    movel(p[new_pose[0], new_pose[1], new_pose[2], current_pose[3], current_pose[4], current_pose[5]], a=1.2, v=0.2000)
    report_progress()
    new_pose = pose_trans(tuft_coords, p[0.8015, 0.1579, -0.0020, 0, 0, 0])
    movel(p[new_pose[0], new_pose[1], new_pose[2], current_pose[3], current_pose[4], current_pose[5]], a=0.8, v=0.2000)
    report_progress()
    set_digital_out(0, True)
    new_pose = pose_trans(tuft_coords, p[0.8015, 0.8921, -0.0020, 0, 0, 0])
    movel(p[new_pose[0], new_pose[1], new_pose[2], current_pose[3], current_pose[4], current_pose[5]], a=1.2, v=0.0600)
    report_progress()
    set_digital_out(0, False)
    new_pose = pose_trans(tuft_coords, p[0.8015, 0.8921, 0.1500, 0, 0, 0])
    movel(p[new_pose[0], new_pose[1], new_pose[2], current_pose[3], current_pose[4], current_pose[5]], a=0.8, v=0.2000)
    report_progress()
    new_pose = pose_trans(tuft_coords, p[0.8035, 0.1579, 0.1500, 0, 0, 0])
    movel(p[new_pose[0], new_pose[1], new_pose[2], current_pose[3], current_pose[4], current_pose[5]], a=1.2, v=0.2000)
    report_progress()
    new_pose = pose_trans(tuft_coords, p[0.8035, 0.1579, -0.0020, 0, 0, 0])
    movel(p[new_pose[0], new_pose[1], new_pose[2], current_pose[3], current_pose[4], current_pose[5]], a=0.8, v=0.2000)
    report_progress()
    set_digital_out(0, True)
    new_pose = pose_trans(tuft_coords, p[0.8035, 0.8921, -0.0020, 0, 0, 0])
    movel(p[new_pose[0], new_pose[1], new_pose[2], current_pose[3], current_pose[4], current_pose[5]], a=1.2, v=0.0600)
    report_progress()
    set_digital_out(0, False)
    new_pose = pose_trans(tuft_coords, p[0.8035, 0.8921, 0.1500, 0, 0, 0])
    movel(p[new_pose[0], new_pose[1], new_pose[2], current_pose[3], current_pose[4], current_pose[5]], a=0.8, v=0.2000)
    report_progress()
    new_pose = pose_trans(tuft_coords, p[0.8054, 0.1579, 0.1500, 0, 0, 0])
    movel(p[new_pose[0], new_pose[1], new_pose[2], current_pose[3], current_pose[4], current_pose[5]], a=1.2, v=0.2000)
    report_progress()
    new_pose = pose_trans(tuft_coords, p[0.8054, 0.1579, -0.0020, 0, 0, 0])
    movel(p[new_pose[0], new_pose[1], new_pose[2], current_pose[3], current_pose[4], current_pose[5]], a=0.8, v=0.2000)
    report_progress()
    set_digital_out(0, True)
    new_pose = pose_trans(tuft_coords, p[0.8054, 0.8921, -0.0020, 0, 0, 0])
    movel(p[new_pose[0], new_pose[1], new_pose[2], current_pose[3], current_pose[4], current_pose[5]], a=1.2, v=0.0600)
    report_progress()
    set_digital_out(0, False)
    new_pose = pose_trans(tuft_coords, p[0.8054, 0.8921, 0.1500, 0, 0, 0])
    movel(p[new_pose[0], new_pose[1], new_pose[2], current_pose[3], current_pose[4], current_pose[5]], a=0.8, v=0.2000)
    report_progress()
    new_pose = pose_trans(tuft_coords, p[0.8074, 0.1598, 0.1500, 0, 0, 0])
    movel(p[new_pose[0], new_pose[1], new_pose[2], current_pose[3], current_pose[4], current_pose[5]], a=1.2, v=0.2000)
    report_progress()
    new_pose = pose_trans(tuft_coords, p[0.8074, 0.1598, -0.0020, 0, 0, 0])
    movel(p[new_pose[0], new_pose[1], new_pose[2], current_pose[3], current_pose[4], current_pose[5]], a=0.8, v=0.2000)
    report_progress()
    set_digital_out(0, True)
    new_pose = pose_trans(tuft_coords, p[0.8074, 0.8902, -0.0020, 0, 0, 0])
    movel(p[new_pose[0], new_pose[1], new_pose[2], current_pose[3], current_pose[4], current_pose[5]], a=1.2, v=0.0600)
    report_progress()
    set_digital_out(0, False)
    new_pose = pose_trans(tuft_coords, p[0.8074, 0.8902, 0.1500, 0, 0, 0])
    movel(p[new_pose[0], new_pose[1], new_pose[2], current_pose[3], current_pose[4], current_pose[5]], a=0.8, v=0.2000)
    report_progress()
    new_pose = pose_trans(tuft_coords, p[0.8093, 0.1598, 0.1500, 0, 0, 0])
    movel(p[new_pose[0], new_pose[1], new_pose[2], current_pose[3], current_pose[4], current_pose[5]], a=1.2, v=0.2000)
    report_progress()
    new_pose = pose_trans(tuft_coords, p[0.8093, 0.1598, -0.0020, 0, 0, 0])
    movel(p[new_pose[0], new_pose[1], new_pose[2], current_pose[3], current_pose[4], current_pose[5]], a=0.8, v=0.2000)
    report_progress()
    set_digital_out(0, True)
    new_pose = pose_trans(tuft_coords, p[0.8093, 0.8902, -0.0020, 0, 0, 0])
    movel(p[new_pose[0], new_pose[1], new_pose[2], current_pose[3], current_pose[4], current_pose[5]], a=1.2, v=0.0600)
    report_progress()
    set_digital_out(0, False)
    new_pose = pose_trans(tuft_coords, p[0.8093, 0.8902, 0.1500, 0, 0, 0])
    movel(p[new_pose[0], new_pose[1], new_pose[2], current_pose[3], current_pose[4], current_pose[5]], a=0.8, v=0.2000)
    report_progress()
    new_pose = pose_trans(tuft_coords, p[0.8113, 0.1598, 0.1500, 0, 0, 0])
    movel(p[new_pose[0], new_pose[1], new_pose[2], current_pose[3], current_pose[4], current_pose[5]], a=1.2, v=0.2000)
    report_progress()
    new_pose = pose_trans(tuft_coords, p[0.8113, 0.1598, -0.0020, 0, 0, 0])
    movel(p[new_pose[0], new_pose[1], new_pose[2], current_pose[3], current_pose[4], current_pose[5]], a=0.8, v=0.2000)
    report_progress()
    set_digital_out(0, True)
    new_pose = pose_trans(tuft_coords, p[0.8113, 0.8902, -0.0020, 0, 0, 0])
    movel(p[new_pose[0], new_pose[1], new_pose[2], current_pose[3], current_pose[4], current_pose[5]], a=1.2, v=0.0600)
    report_progress()
    set_digital_out(0, False)
    new_pose = pose_trans(tuft_coords, p[0.8113, 0.8902, 0.1500, 0, 0, 0])
    movel(p[new_pose[0], new_pose[1], new_pose[2], current_pose[3], current_pose[4], current_pose[5]], a=0.8, v=0.2000)
    report_progress()
    new_pose = pose_trans(tuft_coords, p[0.8132, 0.1598, 0.1500, 0, 0, 0])
    movel(p[new_pose[0], new_pose[1], new_pose[2], current_pose[3], current_pose[4], current_pose[5]], a=1.2, v=0.2000)
    report_progress()
    new_pose = pose_trans(tuft_coords, p[0.8132, 0.1598, -0.0020, 0, 0, 0])
    movel(p[new_pose[0], new_pose[1], new_pose[2], current_pose[3], current_pose[4], current_pose[5]], a=0.8, v=0.2000)
    report_progress()
    set_digital_out(0, True)
    new_pose = pose_trans(tuft_coords, p[0.8132, 0.8902, -0.0020, 0, 0, 0])
    movel(p[new_pose[0], new_pose[1], new_pose[2], current_pose[3], current_pose[4], current_pose[5]], a=1.2, v=0.0600)
    report_progress()
    set_digital_out(0, False)
    new_pose = pose_trans(tuft_coords, p[0.8132, 0.8902, 0.1500, 0, 0, 0])
    movel(p[new_pose[0], new_pose[1], new_pose[2], current_pose[3], current_pose[4], current_pose[5]], a=0.8, v=0.2000)
    report_progress()
    new_pose = pose_trans(tuft_coords, p[0.8151, 0.1598, 0.1500, 0, 0, 0])
    movel(p[new_pose[0], new_pose[1], new_pose[2], current_pose[3], current_pose[4], current_pose[5]], a=1.2, v=0.2000)
    report_progress()
    new_pose = pose_trans(tuft_coords, p[0.8151, 0.1598, -0.0020, 0, 0, 0])
    movel(p[new_pose[0], new_pose[1], new_pose[2], current_pose[3], current_pose[4], current_pose[5]], a=0.8, v=0.2000)
    report_progress()
    set_digital_out(0, True)
    new_pose = pose_trans(tuft_coords, p[0.8151, 0.8902, -0.0020, 0, 0, 0])
    movel(p[new_pose[0], new_pose[1], new_pose[2], current_pose[3], current_pose[4], current_pose[5]], a=1.2, v=0.0600)
    report_progress()
    set_digital_out(0, False)
    new_pose = pose_trans(tuft_coords, p[0.8151, 0.8902, 0.1500, 0, 0, 0])
    movel(p[new_pose[0], new_pose[1], new_pose[2], current_pose[3], current_pose[4], current_pose[5]], a=0.8, v=0.2000)
    report_progress()
    new_pose = pose_trans(tuft_coords, p[0.8171, 0.1598, 0.1500, 0, 0, 0])
    movel(p[new_pose[0], new_pose[1], new_pose[2], current_pose[3], current_pose[4], current_pose[5]], a=1.2, v=0.2000)
    report_progress()
    new_pose = pose_trans(tuft_coords, p[0.8171, 0.1598, -0.0020, 0, 0, 0])
    movel(p[new_pose[0], new_pose[1], new_pose[2], current_pose[3], current_pose[4], current_pose[5]], a=0.8, v=0.2000)
    report_progress()
    set_digital_out(0, True)
    new_pose = pose_trans(tuft_coords, p[0.8171, 0.8902, -0.0020, 0, 0, 0])
    movel(p[new_pose[0], new_pose[1], new_pose[2], current_pose[3], current_pose[4], current_pose[5]], a=1.2, v=0.0600)
    report_progress()
    set_digital_out(0, False)
    new_pose = pose_trans(tuft_coords, p[0.8171, 0.8902, 0.1500, 0, 0, 0])
    movel(p[new_pose[0], new_pose[1], new_pose[2], current_pose[3], current_pose[4], current_pose[5]], a=0.8, v=0.2000)
    report_progress()
    new_pose = pose_trans(tuft_coords, p[0.8190, 0.1618, 0.1500, 0, 0, 0])
    movel(p[new_pose[0], new_pose[1], new_pose[2], current_pose[3], current_pose[4], current_pose[5]], a=1.2, v=0.2000)
    report_progress()
    new_pose = pose_trans(tuft_coords, p[0.8190, 0.1618, -0.0020, 0, 0, 0])
    movel(p[new_pose[0], new_pose[1], new_pose[2], current_pose[3], current_pose[4], current_pose[5]], a=0.8, v=0.2000)
    report_progress()
    set_digital_out(0, True)
    new_pose = pose_trans(tuft_coords, p[0.8190, 0.8882, -0.0020, 0, 0, 0])
    movel(p[new_pose[0], new_pose[1], new_pose[2], current_pose[3], current_pose[4], current_pose[5]], a=1.2, v=0.0600)
    report_progress()
    set_digital_out(0, False)
    new_pose = pose_trans(tuft_coords, p[0.8190, 0.8882, 0.1500, 0, 0, 0])
    movel(p[new_pose[0], new_pose[1], new_pose[2], current_pose[3], current_pose[4], current_pose[5]], a=0.8, v=0.2000)
    report_progress()
    new_pose = pose_trans(tuft_coords, p[0.8210, 0.1618, 0.1500, 0, 0, 0])
    movel(p[new_pose[0], new_pose[1], new_pose[2], current_pose[3], current_pose[4], current_pose[5]], a=1.2, v=0.2000)
    report_progress()
    new_pose = pose_trans(tuft_coords, p[0.8210, 0.1618, -0.0020, 0, 0, 0])
    movel(p[new_pose[0], new_pose[1], new_pose[2], current_pose[3], current_pose[4], current_pose[5]], a=0.8, v=0.2000)
    report_progress()
    set_digital_out(0, True)
    new_pose = pose_trans(tuft_coords, p[0.8210, 0.8882, -0.0020, 0, 0, 0])
    movel(p[new_pose[0], new_pose[1], new_pose[2], current_pose[3], current_pose[4], current_pose[5]], a=1.2, v=0.0600)
    report_progress()
    set_digital_out(0, False)
    new_pose = pose_trans(tuft_coords, p[0.8210, 0.8882, 0.1500, 0, 0, 0])
    movel(p[new_pose[0], new_pose[1], new_pose[2], current_pose[3], current_pose[4], current_pose[5]], a=0.8, v=0.2000)
    report_progress()
    new_pose = pose_trans(tuft_coords, p[0.8229, 0.1618, 0.1500, 0, 0, 0])
    movel(p[new_pose[0], new_pose[1], new_pose[2], current_pose[3], current_pose[4], current_pose[5]], a=1.2, v=0.2000)
    report_progress()
    new_pose = pose_trans(tuft_coords, p[0.8229, 0.1618, -0.0020, 0, 0, 0])
    movel(p[new_pose[0], new_pose[1], new_pose[2], current_pose[3], current_pose[4], current_pose[5]], a=0.8, v=0.2000)
    report_progress()
    set_digital_out(0, True)
    new_pose = pose_trans(tuft_coords, p[0.8229, 0.8882, -0.0020, 0, 0, 0])
    movel(p[new_pose[0], new_pose[1], new_pose[2], current_pose[3], current_pose[4], current_pose[5]], a=1.2, v=0.0600)
    report_progress()
    set_digital_out(0, False)
    new_pose = pose_trans(tuft_coords, p[0.8229, 0.8882, 0.1500, 0, 0, 0])
    movel(p[new_pose[0], new_pose[1], new_pose[2], current_pose[3], current_pose[4], current_pose[5]], a=0.8, v=0.2000)
    report_progress()
    new_pose = pose_trans(tuft_coords, p[0.8249, 0.1618, 0.1500, 0, 0, 0])
    movel(p[new_pose[0], new_pose[1], new_pose[2], current_pose[3], current_pose[4], current_pose[5]], a=1.2, v=0.2000)
    report_progress()
    new_pose = pose_trans(tuft_coords, p[0.8249, 0.1618, -0.0020, 0, 0, 0])
    movel(p[new_pose[0], new_pose[1], new_pose[2], current_pose[3], current_pose[4], current_pose[5]], a=0.8, v=0.2000)
    report_progress()
    set_digital_out(0, True)
    new_pose = pose_trans(tuft_coords, p[0.8249, 0.8882, -0.0020, 0, 0, 0])
    movel(p[new_pose[0], new_pose[1], new_pose[2], current_pose[3], current_pose[4], current_pose[5]], a=1.2, v=0.0600)
    report_progress()
    set_digital_out(0, False)
    new_pose = pose_trans(tuft_coords, p[0.8249, 0.8882, 0.1500, 0, 0, 0])
    movel(p[new_pose[0], new_pose[1], new_pose[2], current_pose[3], current_pose[4], current_pose[5]], a=0.8, v=0.2000)
    report_progress()
    new_pose = pose_trans(tuft_coords, p[0.8268, 0.1618, 0.1500, 0, 0, 0])
    movel(p[new_pose[0], new_pose[1], new_pose[2], current_pose[3], current_pose[4], current_pose[5]], a=1.2, v=0.2000)
    report_progress()
    new_pose = pose_trans(tuft_coords, p[0.8268, 0.1618, -0.0020, 0, 0, 0])
    movel(p[new_pose[0], new_pose[1], new_pose[2], current_pose[3], current_pose[4], current_pose[5]], a=0.8, v=0.2000)
    report_progress()
    set_digital_out(0, True)
    new_pose = pose_trans(tuft_coords, p[0.8268, 0.8882, -0.0020, 0, 0, 0])
    movel(p[new_pose[0], new_pose[1], new_pose[2], current_pose[3], current_pose[4], current_pose[5]], a=1.2, v=0.0600)
    report_progress()
    set_digital_out(0, False)
    new_pose = pose_trans(tuft_coords, p[0.8268, 0.8882, 0.1500, 0, 0, 0])
    movel(p[new_pose[0], new_pose[1], new_pose[2], current_pose[3], current_pose[4], current_pose[5]], a=0.8, v=0.2000)
    report_progress()
    new_pose = pose_trans(tuft_coords, p[0.8287, 0.1638, 0.1500, 0, 0, 0])
    movel(p[new_pose[0], new_pose[1], new_pose[2], current_pose[3], current_pose[4], current_pose[5]], a=1.2, v=0.2000)
    report_progress()
    new_pose = pose_trans(tuft_coords, p[0.8287, 0.1638, -0.0020, 0, 0, 0])
    movel(p[new_pose[0], new_pose[1], new_pose[2], current_pose[3], current_pose[4], current_pose[5]], a=0.8, v=0.2000)
    report_progress()
    set_digital_out(0, True)
    new_pose = pose_trans(tuft_coords, p[0.8287, 0.8862, -0.0020, 0, 0, 0])
    movel(p[new_pose[0], new_pose[1], new_pose[2], current_pose[3], current_pose[4], current_pose[5]], a=1.2, v=0.0600)
    report_progress()
    set_digital_out(0, False)
    new_pose = pose_trans(tuft_coords, p[0.8287, 0.8862, 0.1500, 0, 0, 0])
    movel(p[new_pose[0], new_pose[1], new_pose[2], current_pose[3], current_pose[4], current_pose[5]], a=0.8, v=0.2000)
    report_progress()
    new_pose = pose_trans(tuft_coords, p[0.8307, 0.1638, 0.1500, 0, 0, 0])
    movel(p[new_pose[0], new_pose[1], new_pose[2], current_pose[3], current_pose[4], current_pose[5]], a=1.2, v=0.2000)
    report_progress()
    new_pose = pose_trans(tuft_coords, p[0.8307, 0.1638, -0.0020, 0, 0, 0])
    movel(p[new_pose[0], new_pose[1], new_pose[2], current_pose[3], current_pose[4], current_pose[5]], a=0.8, v=0.2000)
    report_progress()
    set_digital_out(0, True)
    new_pose = pose_trans(tuft_coords, p[0.8307, 0.8862, -0.0020, 0, 0, 0])
    movel(p[new_pose[0], new_pose[1], new_pose[2], current_pose[3], current_pose[4], current_pose[5]], a=1.2, v=0.0600)
    report_progress()
    set_digital_out(0, False)
    new_pose = pose_trans(tuft_coords, p[0.8307, 0.8862, 0.1500, 0, 0, 0])
    movel(p[new_pose[0], new_pose[1], new_pose[2], current_pose[3], current_pose[4], current_pose[5]], a=0.8, v=0.2000)
    report_progress()
    new_pose = pose_trans(tuft_coords, p[0.8326, 0.1638, 0.1500, 0, 0, 0])
    movel(p[new_pose[0], new_pose[1], new_pose[2], current_pose[3], current_pose[4], current_pose[5]], a=1.2, v=0.2000)
    report_progress()
    new_pose = pose_trans(tuft_coords, p[0.8326, 0.1638, -0.0020, 0, 0, 0])
    movel(p[new_pose[0], new_pose[1], new_pose[2], current_pose[3], current_pose[4], current_pose[5]], a=0.8, v=0.2000)
    report_progress()
    set_digital_out(0, True)
    new_pose = pose_trans(tuft_coords, p[0.8326, 0.8862, -0.0020, 0, 0, 0])
    movel(p[new_pose[0], new_pose[1], new_pose[2], current_pose[3], current_pose[4], current_pose[5]], a=1.2, v=0.0600)
    report_progress()
    set_digital_out(0, False)
    new_pose = pose_trans(tuft_coords, p[0.8326, 0.8862, 0.1500, 0, 0, 0])
    movel(p[new_pose[0], new_pose[1], new_pose[2], current_pose[3], current_pose[4], current_pose[5]], a=0.8, v=0.2000)
    report_progress()
    new_pose = pose_trans(tuft_coords, p[0.8346, 0.1638, 0.1500, 0, 0, 0])
    movel(p[new_pose[0], new_pose[1], new_pose[2], current_pose[3], current_pose[4], current_pose[5]], a=1.2, v=0.2000)
    report_progress()
    new_pose = pose_trans(tuft_coords, p[0.8346, 0.1638, -0.0020, 0, 0, 0])
    movel(p[new_pose[0], new_pose[1], new_pose[2], current_pose[3], current_pose[4], current_pose[5]], a=0.8, v=0.2000)
    report_progress()
    set_digital_out(0, True)
    new_pose = pose_trans(tuft_coords, p[0.8346, 0.8862, -0.0020, 0, 0, 0])
    movel(p[new_pose[0], new_pose[1], new_pose[2], current_pose[3], current_pose[4], current_pose[5]], a=1.2, v=0.0600)
    report_progress()
    set_digital_out(0, False)
    new_pose = pose_trans(tuft_coords, p[0.8346, 0.8862, 0.1500, 0, 0, 0])
    movel(p[new_pose[0], new_pose[1], new_pose[2], current_pose[3], current_pose[4], current_pose[5]], a=0.8, v=0.2000)
    report_progress()
    new_pose = pose_trans(tuft_coords, p[0.8365, 0.1658, 0.1500, 0, 0, 0])
    movel(p[new_pose[0], new_pose[1], new_pose[2], current_pose[3], current_pose[4], current_pose[5]], a=1.2, v=0.2000)
    report_progress()
    new_pose = pose_trans(tuft_coords, p[0.8365, 0.1658, -0.0020, 0, 0, 0])
    movel(p[new_pose[0], new_pose[1], new_pose[2], current_pose[3], current_pose[4], current_pose[5]], a=0.8, v=0.2000)
    report_progress()
    set_digital_out(0, True)
    new_pose = pose_trans(tuft_coords, p[0.8365, 0.8842, -0.0020, 0, 0, 0])
    movel(p[new_pose[0], new_pose[1], new_pose[2], current_pose[3], current_pose[4], current_pose[5]], a=1.2, v=0.0600)
    report_progress()
    set_digital_out(0, False)
    new_pose = pose_trans(tuft_coords, p[0.8365, 0.8842, 0.1500, 0, 0, 0])
    movel(p[new_pose[0], new_pose[1], new_pose[2], current_pose[3], current_pose[4], current_pose[5]], a=0.8, v=0.2000)
    report_progress()
    new_pose = pose_trans(tuft_coords, p[0.8385, 0.1658, 0.1500, 0, 0, 0])
    movel(p[new_pose[0], new_pose[1], new_pose[2], current_pose[3], current_pose[4], current_pose[5]], a=1.2, v=0.2000)
    report_progress()
    new_pose = pose_trans(tuft_coords, p[0.8385, 0.1658, -0.0020, 0, 0, 0])
    movel(p[new_pose[0], new_pose[1], new_pose[2], current_pose[3], current_pose[4], current_pose[5]], a=0.8, v=0.2000)
    report_progress()
    set_digital_out(0, True)
    new_pose = pose_trans(tuft_coords, p[0.8385, 0.8842, -0.0020, 0, 0, 0])
    movel(p[new_pose[0], new_pose[1], new_pose[2], current_pose[3], current_pose[4], current_pose[5]], a=1.2, v=0.0600)
    report_progress()
    set_digital_out(0, False)
    new_pose = pose_trans(tuft_coords, p[0.8385, 0.8842, 0.1500, 0, 0, 0])
    movel(p[new_pose[0], new_pose[1], new_pose[2], current_pose[3], current_pose[4], current_pose[5]], a=0.8, v=0.2000)
    report_progress()
    new_pose = pose_trans(tuft_coords, p[0.8404, 0.1658, 0.1500, 0, 0, 0])
    movel(p[new_pose[0], new_pose[1], new_pose[2], current_pose[3], current_pose[4], current_pose[5]], a=1.2, v=0.2000)
    report_progress()
    new_pose = pose_trans(tuft_coords, p[0.8404, 0.1658, -0.0020, 0, 0, 0])
    movel(p[new_pose[0], new_pose[1], new_pose[2], current_pose[3], current_pose[4], current_pose[5]], a=0.8, v=0.2000)
    report_progress()
    set_digital_out(0, True)
    new_pose = pose_trans(tuft_coords, p[0.8404, 0.8842, -0.0020, 0, 0, 0])
    movel(p[new_pose[0], new_pose[1], new_pose[2], current_pose[3], current_pose[4], current_pose[5]], a=1.2, v=0.0600)
    report_progress()
    set_digital_out(0, False)
    new_pose = pose_trans(tuft_coords, p[0.8404, 0.8842, 0.1500, 0, 0, 0])
    movel(p[new_pose[0], new_pose[1], new_pose[2], current_pose[3], current_pose[4], current_pose[5]], a=0.8, v=0.2000)
    report_progress()
    new_pose = pose_trans(tuft_coords, p[0.8424, 0.1658, 0.1500, 0, 0, 0])
    movel(p[new_pose[0], new_pose[1], new_pose[2], current_pose[3], current_pose[4], current_pose[5]], a=1.2, v=0.2000)
    report_progress()
    new_pose = pose_trans(tuft_coords, p[0.8424, 0.1658, -0.0020, 0, 0, 0])
    movel(p[new_pose[0], new_pose[1], new_pose[2], current_pose[3], current_pose[4], current_pose[5]], a=0.8, v=0.2000)
    report_progress()
    set_digital_out(0, True)
    new_pose = pose_trans(tuft_coords, p[0.8424, 0.8842, -0.0020, 0, 0, 0])
    movel(p[new_pose[0], new_pose[1], new_pose[2], current_pose[3], current_pose[4], current_pose[5]], a=1.2, v=0.0600)
    report_progress()
    set_digital_out(0, False)
    new_pose = pose_trans(tuft_coords, p[0.8424, 0.8842, 0.1500, 0, 0, 0])
    movel(p[new_pose[0], new_pose[1], new_pose[2], current_pose[3], current_pose[4], current_pose[5]], a=0.8, v=0.2000)
    report_progress()
    new_pose = pose_trans(tuft_coords, p[0.8443, 0.1678, 0.1500, 0, 0, 0])
    movel(p[new_pose[0], new_pose[1], new_pose[2], current_pose[3], current_pose[4], current_pose[5]], a=1.2, v=0.2000)
    report_progress()
    new_pose = pose_trans(tuft_coords, p[0.8443, 0.1678, -0.0020, 0, 0, 0])
    movel(p[new_pose[0], new_pose[1], new_pose[2], current_pose[3], current_pose[4], current_pose[5]], a=0.8, v=0.2000)
    report_progress()
    set_digital_out(0, True)
    new_pose = pose_trans(tuft_coords, p[0.8443, 0.8822, -0.0020, 0, 0, 0])
    movel(p[new_pose[0], new_pose[1], new_pose[2], current_pose[3], current_pose[4], current_pose[5]], a=1.2, v=0.0600)
    report_progress()
    set_digital_out(0, False)
    new_pose = pose_trans(tuft_coords, p[0.8443, 0.8822, 0.1500, 0, 0, 0])
    movel(p[new_pose[0], new_pose[1], new_pose[2], current_pose[3], current_pose[4], current_pose[5]], a=0.8, v=0.2000)
    report_progress()
    new_pose = pose_trans(tuft_coords, p[0.8462, 0.1678, 0.1500, 0, 0, 0])
    movel(p[new_pose[0], new_pose[1], new_pose[2], current_pose[3], current_pose[4], current_pose[5]], a=1.2, v=0.2000)
    report_progress()
    new_pose = pose_trans(tuft_coords, p[0.8462, 0.1678, -0.0020, 0, 0, 0])
    movel(p[new_pose[0], new_pose[1], new_pose[2], current_pose[3], current_pose[4], current_pose[5]], a=0.8, v=0.2000)
    report_progress()
    set_digital_out(0, True)
    new_pose = pose_trans(tuft_coords, p[0.8462, 0.8822, -0.0020, 0, 0, 0])
    movel(p[new_pose[0], new_pose[1], new_pose[2], current_pose[3], current_pose[4], current_pose[5]], a=1.2, v=0.0600)
    report_progress()
    set_digital_out(0, False)
    new_pose = pose_trans(tuft_coords, p[0.8462, 0.8822, 0.1500, 0, 0, 0])
    movel(p[new_pose[0], new_pose[1], new_pose[2], current_pose[3], current_pose[4], current_pose[5]], a=0.8, v=0.2000)
    report_progress()
    new_pose = pose_trans(tuft_coords, p[0.8482, 0.1678, 0.1500, 0, 0, 0])
    movel(p[new_pose[0], new_pose[1], new_pose[2], current_pose[3], current_pose[4], current_pose[5]], a=1.2, v=0.2000)
    report_progress()
    new_pose = pose_trans(tuft_coords, p[0.8482, 0.1678, -0.0020, 0, 0, 0])
    movel(p[new_pose[0], new_pose[1], new_pose[2], current_pose[3], current_pose[4], current_pose[5]], a=0.8, v=0.2000)
    report_progress()
    set_digital_out(0, True)
    new_pose = pose_trans(tuft_coords, p[0.8482, 0.8822, -0.0020, 0, 0, 0])
    movel(p[new_pose[0], new_pose[1], new_pose[2], current_pose[3], current_pose[4], current_pose[5]], a=1.2, v=0.0600)
    report_progress()
    set_digital_out(0, False)
    new_pose = pose_trans(tuft_coords, p[0.8482, 0.8822, 0.1500, 0, 0, 0])
    movel(p[new_pose[0], new_pose[1], new_pose[2], current_pose[3], current_pose[4], current_pose[5]], a=0.8, v=0.2000)
    report_progress()
    new_pose = pose_trans(tuft_coords, p[0.8501, 0.1678, 0.1500, 0, 0, 0])
    movel(p[new_pose[0], new_pose[1], new_pose[2], current_pose[3], current_pose[4], current_pose[5]], a=1.2, v=0.2000)
    report_progress()
    new_pose = pose_trans(tuft_coords, p[0.8501, 0.1678, -0.0020, 0, 0, 0])
    movel(p[new_pose[0], new_pose[1], new_pose[2], current_pose[3], current_pose[4], current_pose[5]], a=0.8, v=0.2000)
    report_progress()
    set_digital_out(0, True)
    new_pose = pose_trans(tuft_coords, p[0.8501, 0.8822, -0.0020, 0, 0, 0])
    movel(p[new_pose[0], new_pose[1], new_pose[2], current_pose[3], current_pose[4], current_pose[5]], a=1.2, v=0.0600)
    report_progress()
    set_digital_out(0, False)
    new_pose = pose_trans(tuft_coords, p[0.8501, 0.8822, 0.1500, 0, 0, 0])
    movel(p[new_pose[0], new_pose[1], new_pose[2], current_pose[3], current_pose[4], current_pose[5]], a=0.8, v=0.2000)
    report_progress()
    new_pose = pose_trans(tuft_coords, p[0.8521, 0.1697, 0.1500, 0, 0, 0])
    movel(p[new_pose[0], new_pose[1], new_pose[2], current_pose[3], current_pose[4], current_pose[5]], a=1.2, v=0.2000)
    report_progress()
    new_pose = pose_trans(tuft_coords, p[0.8521, 0.1697, -0.0020, 0, 0, 0])
    movel(p[new_pose[0], new_pose[1], new_pose[2], current_pose[3], current_pose[4], current_pose[5]], a=0.8, v=0.2000)
    report_progress()
    set_digital_out(0, True)
    new_pose = pose_trans(tuft_coords, p[0.8521, 0.8803, -0.0020, 0, 0, 0])
    movel(p[new_pose[0], new_pose[1], new_pose[2], current_pose[3], current_pose[4], current_pose[5]], a=1.2, v=0.0600)
    report_progress()
    set_digital_out(0, False)
    new_pose = pose_trans(tuft_coords, p[0.8521, 0.8803, 0.1500, 0, 0, 0])
    movel(p[new_pose[0], new_pose[1], new_pose[2], current_pose[3], current_pose[4], current_pose[5]], a=0.8, v=0.2000)
    report_progress()
    new_pose = pose_trans(tuft_coords, p[0.8540, 0.1697, 0.1500, 0, 0, 0])
    movel(p[new_pose[0], new_pose[1], new_pose[2], current_pose[3], current_pose[4], current_pose[5]], a=1.2, v=0.2000)
    report_progress()
    new_pose = pose_trans(tuft_coords, p[0.8540, 0.1697, -0.0020, 0, 0, 0])
    movel(p[new_pose[0], new_pose[1], new_pose[2], current_pose[3], current_pose[4], current_pose[5]], a=0.8, v=0.2000)
    report_progress()
    set_digital_out(0, True)
    new_pose = pose_trans(tuft_coords, p[0.8540, 0.8803, -0.0020, 0, 0, 0])
    movel(p[new_pose[0], new_pose[1], new_pose[2], current_pose[3], current_pose[4], current_pose[5]], a=1.2, v=0.0600)
    report_progress()
    set_digital_out(0, False)
    new_pose = pose_trans(tuft_coords, p[0.8540, 0.8803, 0.1500, 0, 0, 0])
    movel(p[new_pose[0], new_pose[1], new_pose[2], current_pose[3], current_pose[4], current_pose[5]], a=0.8, v=0.2000)
    report_progress()
    new_pose = pose_trans(tuft_coords, p[0.8560, 0.1697, 0.1500, 0, 0, 0])
    movel(p[new_pose[0], new_pose[1], new_pose[2], current_pose[3], current_pose[4], current_pose[5]], a=1.2, v=0.2000)
    report_progress()
    new_pose = pose_trans(tuft_coords, p[0.8560, 0.1697, -0.0020, 0, 0, 0])
    movel(p[new_pose[0], new_pose[1], new_pose[2], current_pose[3], current_pose[4], current_pose[5]], a=0.8, v=0.2000)
    report_progress()
    set_digital_out(0, True)
    new_pose = pose_trans(tuft_coords, p[0.8560, 0.8803, -0.0020, 0, 0, 0])
    movel(p[new_pose[0], new_pose[1], new_pose[2], current_pose[3], current_pose[4], current_pose[5]], a=1.2, v=0.0600)
    report_progress()
    set_digital_out(0, False)
    new_pose = pose_trans(tuft_coords, p[0.8560, 0.8803, 0.1500, 0, 0, 0])
    movel(p[new_pose[0], new_pose[1], new_pose[2], current_pose[3], current_pose[4], current_pose[5]], a=0.8, v=0.2000)
    report_progress()
    new_pose = pose_trans(tuft_coords, p[0.8579, 0.1717, 0.1500, 0, 0, 0])
    movel(p[new_pose[0], new_pose[1], new_pose[2], current_pose[3], current_pose[4], current_pose[5]], a=1.2, v=0.2000)
    report_progress()
    new_pose = pose_trans(tuft_coords, p[0.8579, 0.1717, -0.0020, 0, 0, 0])
    movel(p[new_pose[0], new_pose[1], new_pose[2], current_pose[3], current_pose[4], current_pose[5]], a=0.8, v=0.2000)
    report_progress()
    set_digital_out(0, True)
    new_pose = pose_trans(tuft_coords, p[0.8579, 0.8783, -0.0020, 0, 0, 0])
    movel(p[new_pose[0], new_pose[1], new_pose[2], current_pose[3], current_pose[4], current_pose[5]], a=1.2, v=0.0600)
    report_progress()
    set_digital_out(0, False)
    new_pose = pose_trans(tuft_coords, p[0.8579, 0.8783, 0.1500, 0, 0, 0])
    movel(p[new_pose[0], new_pose[1], new_pose[2], current_pose[3], current_pose[4], current_pose[5]], a=0.8, v=0.2000)
    report_progress()
    new_pose = pose_trans(tuft_coords, p[0.8599, 0.1717, 0.1500, 0, 0, 0])
    movel(p[new_pose[0], new_pose[1], new_pose[2], current_pose[3], current_pose[4], current_pose[5]], a=1.2, v=0.2000)
    report_progress()
    new_pose = pose_trans(tuft_coords, p[0.8599, 0.1717, -0.0020, 0, 0, 0])
    movel(p[new_pose[0], new_pose[1], new_pose[2], current_pose[3], current_pose[4], current_pose[5]], a=0.8, v=0.2000)
    report_progress()
    set_digital_out(0, True)
    new_pose = pose_trans(tuft_coords, p[0.8599, 0.8783, -0.0020, 0, 0, 0])
    movel(p[new_pose[0], new_pose[1], new_pose[2], current_pose[3], current_pose[4], current_pose[5]], a=1.2, v=0.0600)
    report_progress()
    set_digital_out(0, False)
    new_pose = pose_trans(tuft_coords, p[0.8599, 0.8783, 0.1500, 0, 0, 0])
    movel(p[new_pose[0], new_pose[1], new_pose[2], current_pose[3], current_pose[4], current_pose[5]], a=0.8, v=0.2000)
    report_progress()
    new_pose = pose_trans(tuft_coords, p[0.8618, 0.1717, 0.1500, 0, 0, 0])
    movel(p[new_pose[0], new_pose[1], new_pose[2], current_pose[3], current_pose[4], current_pose[5]], a=1.2, v=0.2000)
    report_progress()
    new_pose = pose_trans(tuft_coords, p[0.8618, 0.1717, -0.0020, 0, 0, 0])
    movel(p[new_pose[0], new_pose[1], new_pose[2], current_pose[3], current_pose[4], current_pose[5]], a=0.8, v=0.2000)
    report_progress()
    set_digital_out(0, True)
    new_pose = pose_trans(tuft_coords, p[0.8618, 0.8783, -0.0020, 0, 0, 0])
    movel(p[new_pose[0], new_pose[1], new_pose[2], current_pose[3], current_pose[4], current_pose[5]], a=1.2, v=0.0600)
    report_progress()
    set_digital_out(0, False)
    new_pose = pose_trans(tuft_coords, p[0.8618, 0.8783, 0.1500, 0, 0, 0])
    movel(p[new_pose[0], new_pose[1], new_pose[2], current_pose[3], current_pose[4], current_pose[5]], a=0.8, v=0.2000)
    report_progress()
    new_pose = pose_trans(tuft_coords, p[0.8638, 0.1737, 0.1500, 0, 0, 0])
    movel(p[new_pose[0], new_pose[1], new_pose[2], current_pose[3], current_pose[4], current_pose[5]], a=1.2, v=0.2000)
    report_progress()
    new_pose = pose_trans(tuft_coords, p[0.8638, 0.1737, -0.0020, 0, 0, 0])
    movel(p[new_pose[0], new_pose[1], new_pose[2], current_pose[3], current_pose[4], current_pose[5]], a=0.8, v=0.2000)
    report_progress()
    set_digital_out(0, True)
    new_pose = pose_trans(tuft_coords, p[0.8638, 0.8763, -0.0020, 0, 0, 0])
    movel(p[new_pose[0], new_pose[1], new_pose[2], current_pose[3], current_pose[4], current_pose[5]], a=1.2, v=0.0600)
    report_progress()
    set_digital_out(0, False)
    new_pose = pose_trans(tuft_coords, p[0.8638, 0.8763, 0.1500, 0, 0, 0])
    movel(p[new_pose[0], new_pose[1], new_pose[2], current_pose[3], current_pose[4], current_pose[5]], a=0.8, v=0.2000)
    report_progress()
    new_pose = pose_trans(tuft_coords, p[0.8657, 0.1737, 0.1500, 0, 0, 0])
    movel(p[new_pose[0], new_pose[1], new_pose[2], current_pose[3], current_pose[4], current_pose[5]], a=1.2, v=0.2000)
    report_progress()
    new_pose = pose_trans(tuft_coords, p[0.8657, 0.1737, -0.0020, 0, 0, 0])
    movel(p[new_pose[0], new_pose[1], new_pose[2], current_pose[3], current_pose[4], current_pose[5]], a=0.8, v=0.2000)
    report_progress()
    set_digital_out(0, True)
    new_pose = pose_trans(tuft_coords, p[0.8657, 0.8763, -0.0020, 0, 0, 0])
    movel(p[new_pose[0], new_pose[1], new_pose[2], current_pose[3], current_pose[4], current_pose[5]], a=1.2, v=0.0600)
    report_progress()
    set_digital_out(0, False)
    new_pose = pose_trans(tuft_coords, p[0.8657, 0.8763, 0.1500, 0, 0, 0])
    movel(p[new_pose[0], new_pose[1], new_pose[2], current_pose[3], current_pose[4], current_pose[5]], a=0.8, v=0.2000)
    report_progress()
    new_pose = pose_trans(tuft_coords, p[0.8676, 0.1737, 0.1500, 0, 0, 0])
    movel(p[new_pose[0], new_pose[1], new_pose[2], current_pose[3], current_pose[4], current_pose[5]], a=1.2, v=0.2000)
    report_progress()
    new_pose = pose_trans(tuft_coords, p[0.8676, 0.1737, -0.0020, 0, 0, 0])
    movel(p[new_pose[0], new_pose[1], new_pose[2], current_pose[3], current_pose[4], current_pose[5]], a=0.8, v=0.2000)
    report_progress()
    set_digital_out(0, True)
    new_pose = pose_trans(tuft_coords, p[0.8676, 0.8763, -0.0020, 0, 0, 0])
    movel(p[new_pose[0], new_pose[1], new_pose[2], current_pose[3], current_pose[4], current_pose[5]], a=1.2, v=0.0600)
    report_progress()
    set_digital_out(0, False)
    new_pose = pose_trans(tuft_coords, p[0.8676, 0.8763, 0.1500, 0, 0, 0])
    movel(p[new_pose[0], new_pose[1], new_pose[2], current_pose[3], current_pose[4], current_pose[5]], a=0.8, v=0.2000)
    report_progress()
    new_pose = pose_trans(tuft_coords, p[0.8696, 0.1757, 0.1500, 0, 0, 0])
    movel(p[new_pose[0], new_pose[1], new_pose[2], current_pose[3], current_pose[4], current_pose[5]], a=1.2, v=0.2000)
    report_progress()
    new_pose = pose_trans(tuft_coords, p[0.8696, 0.1757, -0.0020, 0, 0, 0])
    movel(p[new_pose[0], new_pose[1], new_pose[2], current_pose[3], current_pose[4], current_pose[5]], a=0.8, v=0.2000)
    report_progress()
    set_digital_out(0, True)
    new_pose = pose_trans(tuft_coords, p[0.8696, 0.8743, -0.0020, 0, 0, 0])
    movel(p[new_pose[0], new_pose[1], new_pose[2], current_pose[3], current_pose[4], current_pose[5]], a=1.2, v=0.0600)
    report_progress()
    set_digital_out(0, False)
    new_pose = pose_trans(tuft_coords, p[0.8696, 0.8743, 0.1500, 0, 0, 0])
    movel(p[new_pose[0], new_pose[1], new_pose[2], current_pose[3], current_pose[4], current_pose[5]], a=0.8, v=0.2000)
    report_progress()
    new_pose = pose_trans(tuft_coords, p[0.8715, 0.1757, 0.1500, 0, 0, 0])
    movel(p[new_pose[0], new_pose[1], new_pose[2], current_pose[3], current_pose[4], current_pose[5]], a=1.2, v=0.2000)
    report_progress()
    new_pose = pose_trans(tuft_coords, p[0.8715, 0.1757, -0.0020, 0, 0, 0])
    movel(p[new_pose[0], new_pose[1], new_pose[2], current_pose[3], current_pose[4], current_pose[5]], a=0.8, v=0.2000)
    report_progress()
    set_digital_out(0, True)
    new_pose = pose_trans(tuft_coords, p[0.8715, 0.8743, -0.0020, 0, 0, 0])
    movel(p[new_pose[0], new_pose[1], new_pose[2], current_pose[3], current_pose[4], current_pose[5]], a=1.2, v=0.0600)
    report_progress()
    set_digital_out(0, False)
    new_pose = pose_trans(tuft_coords, p[0.8715, 0.8743, 0.1500, 0, 0, 0])
    movel(p[new_pose[0], new_pose[1], new_pose[2], current_pose[3], current_pose[4], current_pose[5]], a=0.8, v=0.2000)
    report_progress()
    new_pose = pose_trans(tuft_coords, p[0.8735, 0.1757, 0.1500, 0, 0, 0])
    movel(p[new_pose[0], new_pose[1], new_pose[2], current_pose[3], current_pose[4], current_pose[5]], a=1.2, v=0.2000)
    report_progress()
    new_pose = pose_trans(tuft_coords, p[0.8735, 0.1757, -0.0020, 0, 0, 0])
    movel(p[new_pose[0], new_pose[1], new_pose[2], current_pose[3], current_pose[4], current_pose[5]], a=0.8, v=0.2000)
    report_progress()
    set_digital_out(0, True)
    new_pose = pose_trans(tuft_coords, p[0.8735, 0.8743, -0.0020, 0, 0, 0])
    movel(p[new_pose[0], new_pose[1], new_pose[2], current_pose[3], current_pose[4], current_pose[5]], a=1.2, v=0.0600)
    report_progress()
    set_digital_out(0, False)
    new_pose = pose_trans(tuft_coords, p[0.8735, 0.8743, 0.1500, 0, 0, 0])
    movel(p[new_pose[0], new_pose[1], new_pose[2], current_pose[3], current_pose[4], current_pose[5]], a=0.8, v=0.2000)
    report_progress()
    new_pose = pose_trans(tuft_coords, p[0.8754, 0.1777, 0.1500, 0, 0, 0])
    movel(p[new_pose[0], new_pose[1], new_pose[2], current_pose[3], current_pose[4], current_pose[5]], a=1.2, v=0.2000)
    report_progress()
    new_pose = pose_trans(tuft_coords, p[0.8754, 0.1777, -0.0020, 0, 0, 0])
    movel(p[new_pose[0], new_pose[1], new_pose[2], current_pose[3], current_pose[4], current_pose[5]], a=0.8, v=0.2000)
    report_progress()
    set_digital_out(0, True)
    new_pose = pose_trans(tuft_coords, p[0.8754, 0.8723, -0.0020, 0, 0, 0])
    movel(p[new_pose[0], new_pose[1], new_pose[2], current_pose[3], current_pose[4], current_pose[5]], a=1.2, v=0.0600)
    report_progress()
    set_digital_out(0, False)
    new_pose = pose_trans(tuft_coords, p[0.8754, 0.8723, 0.1500, 0, 0, 0])
    movel(p[new_pose[0], new_pose[1], new_pose[2], current_pose[3], current_pose[4], current_pose[5]], a=0.8, v=0.2000)
    report_progress()
    new_pose = pose_trans(tuft_coords, p[0.8774, 0.1777, 0.1500, 0, 0, 0])
    movel(p[new_pose[0], new_pose[1], new_pose[2], current_pose[3], current_pose[4], current_pose[5]], a=1.2, v=0.2000)
    report_progress()
    new_pose = pose_trans(tuft_coords, p[0.8774, 0.1777, -0.0020, 0, 0, 0])
    movel(p[new_pose[0], new_pose[1], new_pose[2], current_pose[3], current_pose[4], current_pose[5]], a=0.8, v=0.2000)
    report_progress()
    set_digital_out(0, True)
    new_pose = pose_trans(tuft_coords, p[0.8774, 0.8723, -0.0020, 0, 0, 0])
    movel(p[new_pose[0], new_pose[1], new_pose[2], current_pose[3], current_pose[4], current_pose[5]], a=1.2, v=0.0600)
    report_progress()
    set_digital_out(0, False)
    new_pose = pose_trans(tuft_coords, p[0.8774, 0.8723, 0.1500, 0, 0, 0])
    movel(p[new_pose[0], new_pose[1], new_pose[2], current_pose[3], current_pose[4], current_pose[5]], a=0.8, v=0.2000)
    report_progress()
    new_pose = pose_trans(tuft_coords, p[0.8793, 0.1777, 0.1500, 0, 0, 0])
    movel(p[new_pose[0], new_pose[1], new_pose[2], current_pose[3], current_pose[4], current_pose[5]], a=1.2, v=0.2000)
    report_progress()
    new_pose = pose_trans(tuft_coords, p[0.8793, 0.1777, -0.0020, 0, 0, 0])
    movel(p[new_pose[0], new_pose[1], new_pose[2], current_pose[3], current_pose[4], current_pose[5]], a=0.8, v=0.2000)
    report_progress()
    set_digital_out(0, True)
    new_pose = pose_trans(tuft_coords, p[0.8793, 0.8723, -0.0020, 0, 0, 0])
    movel(p[new_pose[0], new_pose[1], new_pose[2], current_pose[3], current_pose[4], current_pose[5]], a=1.2, v=0.0600)
    report_progress()
    set_digital_out(0, False)
    new_pose = pose_trans(tuft_coords, p[0.8793, 0.8723, 0.1500, 0, 0, 0])
    movel(p[new_pose[0], new_pose[1], new_pose[2], current_pose[3], current_pose[4], current_pose[5]], a=0.8, v=0.2000)
    report_progress()
    new_pose = pose_trans(tuft_coords, p[0.8812, 0.1796, 0.1500, 0, 0, 0])
    movel(p[new_pose[0], new_pose[1], new_pose[2], current_pose[3], current_pose[4], current_pose[5]], a=1.2, v=0.2000)
    report_progress()
    new_pose = pose_trans(tuft_coords, p[0.8812, 0.1796, -0.0020, 0, 0, 0])
    movel(p[new_pose[0], new_pose[1], new_pose[2], current_pose[3], current_pose[4], current_pose[5]], a=0.8, v=0.2000)
    report_progress()
    set_digital_out(0, True)
    new_pose = pose_trans(tuft_coords, p[0.8812, 0.8704, -0.0020, 0, 0, 0])
    movel(p[new_pose[0], new_pose[1], new_pose[2], current_pose[3], current_pose[4], current_pose[5]], a=1.2, v=0.0600)
    report_progress()
    set_digital_out(0, False)
    new_pose = pose_trans(tuft_coords, p[0.8812, 0.8704, 0.1500, 0, 0, 0])
    movel(p[new_pose[0], new_pose[1], new_pose[2], current_pose[3], current_pose[4], current_pose[5]], a=0.8, v=0.2000)
    report_progress()
    new_pose = pose_trans(tuft_coords, p[0.8832, 0.1796, 0.1500, 0, 0, 0])
    movel(p[new_pose[0], new_pose[1], new_pose[2], current_pose[3], current_pose[4], current_pose[5]], a=1.2, v=0.2000)
    report_progress()
    new_pose = pose_trans(tuft_coords, p[0.8832, 0.1796, -0.0020, 0, 0, 0])
    movel(p[new_pose[0], new_pose[1], new_pose[2], current_pose[3], current_pose[4], current_pose[5]], a=0.8, v=0.2000)
    report_progress()
    set_digital_out(0, True)
    new_pose = pose_trans(tuft_coords, p[0.8832, 0.8704, -0.0020, 0, 0, 0])
    movel(p[new_pose[0], new_pose[1], new_pose[2], current_pose[3], current_pose[4], current_pose[5]], a=1.2, v=0.0600)
    report_progress()
    set_digital_out(0, False)
    new_pose = pose_trans(tuft_coords, p[0.8832, 0.8704, 0.1500, 0, 0, 0])
    movel(p[new_pose[0], new_pose[1], new_pose[2], current_pose[3], current_pose[4], current_pose[5]], a=0.8, v=0.2000)
    report_progress()
    new_pose = pose_trans(tuft_coords, p[0.8851, 0.1816, 0.1500, 0, 0, 0])
    movel(p[new_pose[0], new_pose[1], new_pose[2], current_pose[3], current_pose[4], current_pose[5]], a=1.2, v=0.2000)
    report_progress()
    new_pose = pose_trans(tuft_coords, p[0.8851, 0.1816, -0.0020, 0, 0, 0])
    movel(p[new_pose[0], new_pose[1], new_pose[2], current_pose[3], current_pose[4], current_pose[5]], a=0.8, v=0.2000)
    report_progress()
    set_digital_out(0, True)
    new_pose = pose_trans(tuft_coords, p[0.8851, 0.8684, -0.0020, 0, 0, 0])
    movel(p[new_pose[0], new_pose[1], new_pose[2], current_pose[3], current_pose[4], current_pose[5]], a=1.2, v=0.0600)
    report_progress()
    set_digital_out(0, False)
    new_pose = pose_trans(tuft_coords, p[0.8851, 0.8684, 0.1500, 0, 0, 0])
    movel(p[new_pose[0], new_pose[1], new_pose[2], current_pose[3], current_pose[4], current_pose[5]], a=0.8, v=0.2000)
    report_progress()
    new_pose = pose_trans(tuft_coords, p[0.8871, 0.1816, 0.1500, 0, 0, 0])
    movel(p[new_pose[0], new_pose[1], new_pose[2], current_pose[3], current_pose[4], current_pose[5]], a=1.2, v=0.2000)
    report_progress()
    new_pose = pose_trans(tuft_coords, p[0.8871, 0.1816, -0.0020, 0, 0, 0])
    movel(p[new_pose[0], new_pose[1], new_pose[2], current_pose[3], current_pose[4], current_pose[5]], a=0.8, v=0.2000)
    report_progress()
    set_digital_out(0, True)
    new_pose = pose_trans(tuft_coords, p[0.8871, 0.8684, -0.0020, 0, 0, 0])
    movel(p[new_pose[0], new_pose[1], new_pose[2], current_pose[3], current_pose[4], current_pose[5]], a=1.2, v=0.0600)
    report_progress()
    set_digital_out(0, False)
    new_pose = pose_trans(tuft_coords, p[0.8871, 0.8684, 0.1500, 0, 0, 0])
    movel(p[new_pose[0], new_pose[1], new_pose[2], current_pose[3], current_pose[4], current_pose[5]], a=0.8, v=0.2000)
    report_progress()
    new_pose = pose_trans(tuft_coords, p[0.8890, 0.1816, 0.1500, 0, 0, 0])
    movel(p[new_pose[0], new_pose[1], new_pose[2], current_pose[3], current_pose[4], current_pose[5]], a=1.2, v=0.2000)
    report_progress()
    new_pose = pose_trans(tuft_coords, p[0.8890, 0.1816, -0.0020, 0, 0, 0])
    movel(p[new_pose[0], new_pose[1], new_pose[2], current_pose[3], current_pose[4], current_pose[5]], a=0.8, v=0.2000)
    report_progress()
    set_digital_out(0, True)
    new_pose = pose_trans(tuft_coords, p[0.8890, 0.8684, -0.0020, 0, 0, 0])
    movel(p[new_pose[0], new_pose[1], new_pose[2], current_pose[3], current_pose[4], current_pose[5]], a=1.2, v=0.0600)
    report_progress()
    set_digital_out(0, False)
    new_pose = pose_trans(tuft_coords, p[0.8890, 0.8684, 0.1500, 0, 0, 0])
    movel(p[new_pose[0], new_pose[1], new_pose[2], current_pose[3], current_pose[4], current_pose[5]], a=0.8, v=0.2000)
    report_progress()
    new_pose = pose_trans(tuft_coords, p[0.8910, 0.1836, 0.1500, 0, 0, 0])
    movel(p[new_pose[0], new_pose[1], new_pose[2], current_pose[3], current_pose[4], current_pose[5]], a=1.2, v=0.2000)
    report_progress()
    new_pose = pose_trans(tuft_coords, p[0.8910, 0.1836, -0.0020, 0, 0, 0])
    movel(p[new_pose[0], new_pose[1], new_pose[2], current_pose[3], current_pose[4], current_pose[5]], a=0.8, v=0.2000)
    report_progress()
    set_digital_out(0, True)
    new_pose = pose_trans(tuft_coords, p[0.8910, 0.8664, -0.0020, 0, 0, 0])
    movel(p[new_pose[0], new_pose[1], new_pose[2], current_pose[3], current_pose[4], current_pose[5]], a=1.2, v=0.0600)
    report_progress()
    set_digital_out(0, False)
    new_pose = pose_trans(tuft_coords, p[0.8910, 0.8664, 0.1500, 0, 0, 0])
    movel(p[new_pose[0], new_pose[1], new_pose[2], current_pose[3], current_pose[4], current_pose[5]], a=0.8, v=0.2000)
    report_progress()
    new_pose = pose_trans(tuft_coords, p[0.8929, 0.1836, 0.1500, 0, 0, 0])
    movel(p[new_pose[0], new_pose[1], new_pose[2], current_pose[3], current_pose[4], current_pose[5]], a=1.2, v=0.2000)
    report_progress()
    new_pose = pose_trans(tuft_coords, p[0.8929, 0.1836, -0.0020, 0, 0, 0])
    movel(p[new_pose[0], new_pose[1], new_pose[2], current_pose[3], current_pose[4], current_pose[5]], a=0.8, v=0.2000)
    report_progress()
    set_digital_out(0, True)
    new_pose = pose_trans(tuft_coords, p[0.8929, 0.8664, -0.0020, 0, 0, 0])
    movel(p[new_pose[0], new_pose[1], new_pose[2], current_pose[3], current_pose[4], current_pose[5]], a=1.2, v=0.0600)
    report_progress()
    set_digital_out(0, False)
    new_pose = pose_trans(tuft_coords, p[0.8929, 0.8664, 0.1500, 0, 0, 0])
    movel(p[new_pose[0], new_pose[1], new_pose[2], current_pose[3], current_pose[4], current_pose[5]], a=0.8, v=0.2000)
    report_progress()
    new_pose = pose_trans(tuft_coords, p[0.8949, 0.1856, 0.1500, 0, 0, 0])
    movel(p[new_pose[0], new_pose[1], new_pose[2], current_pose[3], current_pose[4], current_pose[5]], a=1.2, v=0.2000)
    report_progress()
    new_pose = pose_trans(tuft_coords, p[0.8949, 0.1856, -0.0020, 0, 0, 0])
    movel(p[new_pose[0], new_pose[1], new_pose[2], current_pose[3], current_pose[4], current_pose[5]], a=0.8, v=0.2000)
    report_progress()
    set_digital_out(0, True)
    new_pose = pose_trans(tuft_coords, p[0.8949, 0.8644, -0.0020, 0, 0, 0])
    movel(p[new_pose[0], new_pose[1], new_pose[2], current_pose[3], current_pose[4], current_pose[5]], a=1.2, v=0.0600)
    report_progress()
    set_digital_out(0, False)
    new_pose = pose_trans(tuft_coords, p[0.8949, 0.8644, 0.1500, 0, 0, 0])
    movel(p[new_pose[0], new_pose[1], new_pose[2], current_pose[3], current_pose[4], current_pose[5]], a=0.8, v=0.2000)
    report_progress()
    new_pose = pose_trans(tuft_coords, p[0.8968, 0.1856, 0.1500, 0, 0, 0])
    movel(p[new_pose[0], new_pose[1], new_pose[2], current_pose[3], current_pose[4], current_pose[5]], a=1.2, v=0.2000)
    report_progress()
    new_pose = pose_trans(tuft_coords, p[0.8968, 0.1856, -0.0020, 0, 0, 0])
    movel(p[new_pose[0], new_pose[1], new_pose[2], current_pose[3], current_pose[4], current_pose[5]], a=0.8, v=0.2000)
    report_progress()
    set_digital_out(0, True)
    new_pose = pose_trans(tuft_coords, p[0.8968, 0.8644, -0.0020, 0, 0, 0])
    movel(p[new_pose[0], new_pose[1], new_pose[2], current_pose[3], current_pose[4], current_pose[5]], a=1.2, v=0.0600)
    report_progress()
    set_digital_out(0, False)
    new_pose = pose_trans(tuft_coords, p[0.8968, 0.8644, 0.1500, 0, 0, 0])
    movel(p[new_pose[0], new_pose[1], new_pose[2], current_pose[3], current_pose[4], current_pose[5]], a=0.8, v=0.2000)
    report_progress()
    new_pose = pose_trans(tuft_coords, p[0.8988, 0.1856, 0.1500, 0, 0, 0])
    movel(p[new_pose[0], new_pose[1], new_pose[2], current_pose[3], current_pose[4], current_pose[5]], a=1.2, v=0.2000)
    report_progress()
    new_pose = pose_trans(tuft_coords, p[0.8988, 0.1856, -0.0020, 0, 0, 0])
    movel(p[new_pose[0], new_pose[1], new_pose[2], current_pose[3], current_pose[4], current_pose[5]], a=0.8, v=0.2000)
    report_progress()
    set_digital_out(0, True)
    new_pose = pose_trans(tuft_coords, p[0.8988, 0.8644, -0.0020, 0, 0, 0])
    movel(p[new_pose[0], new_pose[1], new_pose[2], current_pose[3], current_pose[4], current_pose[5]], a=1.2, v=0.0600)
    report_progress()
    set_digital_out(0, False)
    new_pose = pose_trans(tuft_coords, p[0.8988, 0.8644, 0.1500, 0, 0, 0])
    movel(p[new_pose[0], new_pose[1], new_pose[2], current_pose[3], current_pose[4], current_pose[5]], a=0.8, v=0.2000)
    report_progress()
    new_pose = pose_trans(tuft_coords, p[0.9007, 0.1876, 0.1500, 0, 0, 0])
    movel(p[new_pose[0], new_pose[1], new_pose[2], current_pose[3], current_pose[4], current_pose[5]], a=1.2, v=0.2000)
    report_progress()
    new_pose = pose_trans(tuft_coords, p[0.9007, 0.1876, -0.0020, 0, 0, 0])
    movel(p[new_pose[0], new_pose[1], new_pose[2], current_pose[3], current_pose[4], current_pose[5]], a=0.8, v=0.2000)
    report_progress()
    set_digital_out(0, True)
    new_pose = pose_trans(tuft_coords, p[0.9007, 0.8624, -0.0020, 0, 0, 0])
    movel(p[new_pose[0], new_pose[1], new_pose[2], current_pose[3], current_pose[4], current_pose[5]], a=1.2, v=0.0600)
    report_progress()
    set_digital_out(0, False)
    new_pose = pose_trans(tuft_coords, p[0.9007, 0.8624, 0.1500, 0, 0, 0])
    movel(p[new_pose[0], new_pose[1], new_pose[2], current_pose[3], current_pose[4], current_pose[5]], a=0.8, v=0.2000)
    report_progress()
    new_pose = pose_trans(tuft_coords, p[0.9026, 0.1876, 0.1500, 0, 0, 0])
    movel(p[new_pose[0], new_pose[1], new_pose[2], current_pose[3], current_pose[4], current_pose[5]], a=1.2, v=0.2000)
    report_progress()
    new_pose = pose_trans(tuft_coords, p[0.9026, 0.1876, -0.0020, 0, 0, 0])
    movel(p[new_pose[0], new_pose[1], new_pose[2], current_pose[3], current_pose[4], current_pose[5]], a=0.8, v=0.2000)
    report_progress()
    set_digital_out(0, True)
    new_pose = pose_trans(tuft_coords, p[0.9026, 0.8624, -0.0020, 0, 0, 0])
    movel(p[new_pose[0], new_pose[1], new_pose[2], current_pose[3], current_pose[4], current_pose[5]], a=1.2, v=0.0600)
    report_progress()
    set_digital_out(0, False)
    new_pose = pose_trans(tuft_coords, p[0.9026, 0.8624, 0.1500, 0, 0, 0])
    movel(p[new_pose[0], new_pose[1], new_pose[2], current_pose[3], current_pose[4], current_pose[5]], a=0.8, v=0.2000)
    report_progress()
    new_pose = pose_trans(tuft_coords, p[0.9046, 0.1895, 0.1500, 0, 0, 0])
    movel(p[new_pose[0], new_pose[1], new_pose[2], current_pose[3], current_pose[4], current_pose[5]], a=1.2, v=0.2000)
    report_progress()
    new_pose = pose_trans(tuft_coords, p[0.9046, 0.1895, -0.0020, 0, 0, 0])
    movel(p[new_pose[0], new_pose[1], new_pose[2], current_pose[3], current_pose[4], current_pose[5]], a=0.8, v=0.2000)
    report_progress()
    set_digital_out(0, True)
    new_pose = pose_trans(tuft_coords, p[0.9046, 0.8605, -0.0020, 0, 0, 0])
    movel(p[new_pose[0], new_pose[1], new_pose[2], current_pose[3], current_pose[4], current_pose[5]], a=1.2, v=0.0600)
    report_progress()
    set_digital_out(0, False)
    new_pose = pose_trans(tuft_coords, p[0.9046, 0.8605, 0.1500, 0, 0, 0])
    movel(p[new_pose[0], new_pose[1], new_pose[2], current_pose[3], current_pose[4], current_pose[5]], a=0.8, v=0.2000)
    report_progress()
    new_pose = pose_trans(tuft_coords, p[0.9065, 0.1895, 0.1500, 0, 0, 0])
    movel(p[new_pose[0], new_pose[1], new_pose[2], current_pose[3], current_pose[4], current_pose[5]], a=1.2, v=0.2000)
    report_progress()
    new_pose = pose_trans(tuft_coords, p[0.9065, 0.1895, -0.0020, 0, 0, 0])
    movel(p[new_pose[0], new_pose[1], new_pose[2], current_pose[3], current_pose[4], current_pose[5]], a=0.8, v=0.2000)
    report_progress()
    set_digital_out(0, True)
    new_pose = pose_trans(tuft_coords, p[0.9065, 0.8605, -0.0020, 0, 0, 0])
    movel(p[new_pose[0], new_pose[1], new_pose[2], current_pose[3], current_pose[4], current_pose[5]], a=1.2, v=0.0600)
    report_progress()
    set_digital_out(0, False)
    new_pose = pose_trans(tuft_coords, p[0.9065, 0.8605, 0.1500, 0, 0, 0])
    movel(p[new_pose[0], new_pose[1], new_pose[2], current_pose[3], current_pose[4], current_pose[5]], a=0.8, v=0.2000)
    report_progress()
    new_pose = pose_trans(tuft_coords, p[0.9085, 0.1915, 0.1500, 0, 0, 0])
    movel(p[new_pose[0], new_pose[1], new_pose[2], current_pose[3], current_pose[4], current_pose[5]], a=1.2, v=0.2000)
    report_progress()
    new_pose = pose_trans(tuft_coords, p[0.9085, 0.1915, -0.0020, 0, 0, 0])
    movel(p[new_pose[0], new_pose[1], new_pose[2], current_pose[3], current_pose[4], current_pose[5]], a=0.8, v=0.2000)
    report_progress()
    set_digital_out(0, True)
    new_pose = pose_trans(tuft_coords, p[0.9085, 0.8585, -0.0020, 0, 0, 0])
    movel(p[new_pose[0], new_pose[1], new_pose[2], current_pose[3], current_pose[4], current_pose[5]], a=1.2, v=0.0600)
    report_progress()
    set_digital_out(0, False)
    new_pose = pose_trans(tuft_coords, p[0.9085, 0.8585, 0.1500, 0, 0, 0])
    movel(p[new_pose[0], new_pose[1], new_pose[2], current_pose[3], current_pose[4], current_pose[5]], a=0.8, v=0.2000)
    report_progress()
    new_pose = pose_trans(tuft_coords, p[0.9104, 0.1915, 0.1500, 0, 0, 0])
    movel(p[new_pose[0], new_pose[1], new_pose[2], current_pose[3], current_pose[4], current_pose[5]], a=1.2, v=0.2000)
    report_progress()
    new_pose = pose_trans(tuft_coords, p[0.9104, 0.1915, -0.0020, 0, 0, 0])
    movel(p[new_pose[0], new_pose[1], new_pose[2], current_pose[3], current_pose[4], current_pose[5]], a=0.8, v=0.2000)
    report_progress()
    set_digital_out(0, True)
    new_pose = pose_trans(tuft_coords, p[0.9104, 0.8585, -0.0020, 0, 0, 0])
    movel(p[new_pose[0], new_pose[1], new_pose[2], current_pose[3], current_pose[4], current_pose[5]], a=1.2, v=0.0600)
    report_progress()
    set_digital_out(0, False)
    new_pose = pose_trans(tuft_coords, p[0.9104, 0.8585, 0.1500, 0, 0, 0])
    movel(p[new_pose[0], new_pose[1], new_pose[2], current_pose[3], current_pose[4], current_pose[5]], a=0.8, v=0.2000)
    report_progress()
    new_pose = pose_trans(tuft_coords, p[0.9124, 0.1935, 0.1500, 0, 0, 0])
    movel(p[new_pose[0], new_pose[1], new_pose[2], current_pose[3], current_pose[4], current_pose[5]], a=1.2, v=0.2000)
    report_progress()
    new_pose = pose_trans(tuft_coords, p[0.9124, 0.1935, -0.0020, 0, 0, 0])
    movel(p[new_pose[0], new_pose[1], new_pose[2], current_pose[3], current_pose[4], current_pose[5]], a=0.8, v=0.2000)
    report_progress()
    set_digital_out(0, True)
    new_pose = pose_trans(tuft_coords, p[0.9124, 0.8565, -0.0020, 0, 0, 0])
    movel(p[new_pose[0], new_pose[1], new_pose[2], current_pose[3], current_pose[4], current_pose[5]], a=1.2, v=0.0600)
    report_progress()
    set_digital_out(0, False)
    new_pose = pose_trans(tuft_coords, p[0.9124, 0.8565, 0.1500, 0, 0, 0])
    movel(p[new_pose[0], new_pose[1], new_pose[2], current_pose[3], current_pose[4], current_pose[5]], a=0.8, v=0.2000)
    report_progress()
    new_pose = pose_trans(tuft_coords, p[0.9143, 0.1935, 0.1500, 0, 0, 0])
    movel(p[new_pose[0], new_pose[1], new_pose[2], current_pose[3], current_pose[4], current_pose[5]], a=1.2, v=0.2000)
    report_progress()
    new_pose = pose_trans(tuft_coords, p[0.9143, 0.1935, -0.0020, 0, 0, 0])
    movel(p[new_pose[0], new_pose[1], new_pose[2], current_pose[3], current_pose[4], current_pose[5]], a=0.8, v=0.2000)
    report_progress()
    set_digital_out(0, True)
    new_pose = pose_trans(tuft_coords, p[0.9143, 0.8565, -0.0020, 0, 0, 0])
    movel(p[new_pose[0], new_pose[1], new_pose[2], current_pose[3], current_pose[4], current_pose[5]], a=1.2, v=0.0600)
    report_progress()
    set_digital_out(0, False)
    new_pose = pose_trans(tuft_coords, p[0.9143, 0.8565, 0.1500, 0, 0, 0])
    movel(p[new_pose[0], new_pose[1], new_pose[2], current_pose[3], current_pose[4], current_pose[5]], a=0.8, v=0.2000)
    report_progress()
    new_pose = pose_trans(tuft_coords, p[0.9163, 0.1955, 0.1500, 0, 0, 0])
    movel(p[new_pose[0], new_pose[1], new_pose[2], current_pose[3], current_pose[4], current_pose[5]], a=1.2, v=0.2000)
    report_progress()
    new_pose = pose_trans(tuft_coords, p[0.9163, 0.1955, -0.0020, 0, 0, 0])
    movel(p[new_pose[0], new_pose[1], new_pose[2], current_pose[3], current_pose[4], current_pose[5]], a=0.8, v=0.2000)
    report_progress()
    set_digital_out(0, True)
    new_pose = pose_trans(tuft_coords, p[0.9163, 0.8545, -0.0020, 0, 0, 0])
    movel(p[new_pose[0], new_pose[1], new_pose[2], current_pose[3], current_pose[4], current_pose[5]], a=1.2, v=0.0600)
    report_progress()
    set_digital_out(0, False)
    new_pose = pose_trans(tuft_coords, p[0.9163, 0.8545, 0.1500, 0, 0, 0])
    movel(p[new_pose[0], new_pose[1], new_pose[2], current_pose[3], current_pose[4], current_pose[5]], a=0.8, v=0.2000)
    report_progress()
    new_pose = pose_trans(tuft_coords, p[0.9182, 0.1955, 0.1500, 0, 0, 0])
    movel(p[new_pose[0], new_pose[1], new_pose[2], current_pose[3], current_pose[4], current_pose[5]], a=1.2, v=0.2000)
    report_progress()
    new_pose = pose_trans(tuft_coords, p[0.9182, 0.1955, -0.0020, 0, 0, 0])
    movel(p[new_pose[0], new_pose[1], new_pose[2], current_pose[3], current_pose[4], current_pose[5]], a=0.8, v=0.2000)
    report_progress()
    set_digital_out(0, True)
    new_pose = pose_trans(tuft_coords, p[0.9182, 0.8545, -0.0020, 0, 0, 0])
    movel(p[new_pose[0], new_pose[1], new_pose[2], current_pose[3], current_pose[4], current_pose[5]], a=1.2, v=0.0600)
    report_progress()
    set_digital_out(0, False)
    new_pose = pose_trans(tuft_coords, p[0.9182, 0.8545, 0.1500, 0, 0, 0])
    movel(p[new_pose[0], new_pose[1], new_pose[2], current_pose[3], current_pose[4], current_pose[5]], a=0.8, v=0.2000)
    report_progress()
    new_pose = pose_trans(tuft_coords, p[0.9201, 0.1974, 0.1500, 0, 0, 0])
    movel(p[new_pose[0], new_pose[1], new_pose[2], current_pose[3], current_pose[4], current_pose[5]], a=1.2, v=0.2000)
    report_progress()
    new_pose = pose_trans(tuft_coords, p[0.9201, 0.1974, -0.0020, 0, 0, 0])
    movel(p[new_pose[0], new_pose[1], new_pose[2], current_pose[3], current_pose[4], current_pose[5]], a=0.8, v=0.2000)
    report_progress()
    set_digital_out(0, True)
    new_pose = pose_trans(tuft_coords, p[0.9201, 0.8526, -0.0020, 0, 0, 0])
    movel(p[new_pose[0], new_pose[1], new_pose[2], current_pose[3], current_pose[4], current_pose[5]], a=1.2, v=0.0600)
    report_progress()
    set_digital_out(0, False)
    new_pose = pose_trans(tuft_coords, p[0.9201, 0.8526, 0.1500, 0, 0, 0])
    movel(p[new_pose[0], new_pose[1], new_pose[2], current_pose[3], current_pose[4], current_pose[5]], a=0.8, v=0.2000)
    report_progress()
    new_pose = pose_trans(tuft_coords, p[0.9221, 0.1974, 0.1500, 0, 0, 0])
    movel(p[new_pose[0], new_pose[1], new_pose[2], current_pose[3], current_pose[4], current_pose[5]], a=1.2, v=0.2000)
    report_progress()
    new_pose = pose_trans(tuft_coords, p[0.9221, 0.1974, -0.0020, 0, 0, 0])
    movel(p[new_pose[0], new_pose[1], new_pose[2], current_pose[3], current_pose[4], current_pose[5]], a=0.8, v=0.2000)
    report_progress()
    set_digital_out(0, True)
    new_pose = pose_trans(tuft_coords, p[0.9221, 0.8526, -0.0020, 0, 0, 0])
    movel(p[new_pose[0], new_pose[1], new_pose[2], current_pose[3], current_pose[4], current_pose[5]], a=1.2, v=0.0600)
    report_progress()
    set_digital_out(0, False)
    new_pose = pose_trans(tuft_coords, p[0.9221, 0.8526, 0.1500, 0, 0, 0])
    movel(p[new_pose[0], new_pose[1], new_pose[2], current_pose[3], current_pose[4], current_pose[5]], a=0.8, v=0.2000)
    report_progress()
    new_pose = pose_trans(tuft_coords, p[0.9240, 0.1994, 0.1500, 0, 0, 0])
    movel(p[new_pose[0], new_pose[1], new_pose[2], current_pose[3], current_pose[4], current_pose[5]], a=1.2, v=0.2000)
    report_progress()
    new_pose = pose_trans(tuft_coords, p[0.9240, 0.1994, -0.0020, 0, 0, 0])
    movel(p[new_pose[0], new_pose[1], new_pose[2], current_pose[3], current_pose[4], current_pose[5]], a=0.8, v=0.2000)
    report_progress()
    set_digital_out(0, True)
    new_pose = pose_trans(tuft_coords, p[0.9240, 0.8506, -0.0020, 0, 0, 0])
    movel(p[new_pose[0], new_pose[1], new_pose[2], current_pose[3], current_pose[4], current_pose[5]], a=1.2, v=0.0600)
    report_progress()
    set_digital_out(0, False)
    new_pose = pose_trans(tuft_coords, p[0.9240, 0.8506, 0.1500, 0, 0, 0])
    movel(p[new_pose[0], new_pose[1], new_pose[2], current_pose[3], current_pose[4], current_pose[5]], a=0.8, v=0.2000)
    report_progress()
    new_pose = pose_trans(tuft_coords, p[0.9260, 0.1994, 0.1500, 0, 0, 0])
    movel(p[new_pose[0], new_pose[1], new_pose[2], current_pose[3], current_pose[4], current_pose[5]], a=1.2, v=0.2000)
    report_progress()
    new_pose = pose_trans(tuft_coords, p[0.9260, 0.1994, -0.0020, 0, 0, 0])
    movel(p[new_pose[0], new_pose[1], new_pose[2], current_pose[3], current_pose[4], current_pose[5]], a=0.8, v=0.2000)
    report_progress()
    set_digital_out(0, True)
    new_pose = pose_trans(tuft_coords, p[0.9260, 0.8506, -0.0020, 0, 0, 0])
    movel(p[new_pose[0], new_pose[1], new_pose[2], current_pose[3], current_pose[4], current_pose[5]], a=1.2, v=0.0600)
    report_progress()
    set_digital_out(0, False)
    new_pose = pose_trans(tuft_coords, p[0.9260, 0.8506, 0.1500, 0, 0, 0])
    movel(p[new_pose[0], new_pose[1], new_pose[2], current_pose[3], current_pose[4], current_pose[5]], a=0.8, v=0.2000)
    report_progress()
    new_pose = pose_trans(tuft_coords, p[0.9279, 0.2014, 0.1500, 0, 0, 0])
    movel(p[new_pose[0], new_pose[1], new_pose[2], current_pose[3], current_pose[4], current_pose[5]], a=1.2, v=0.2000)
    report_progress()
    new_pose = pose_trans(tuft_coords, p[0.9279, 0.2014, -0.0020, 0, 0, 0])
    movel(p[new_pose[0], new_pose[1], new_pose[2], current_pose[3], current_pose[4], current_pose[5]], a=0.8, v=0.2000)
    report_progress()
    set_digital_out(0, True)
    new_pose = pose_trans(tuft_coords, p[0.9279, 0.8486, -0.0020, 0, 0, 0])
    movel(p[new_pose[0], new_pose[1], new_pose[2], current_pose[3], current_pose[4], current_pose[5]], a=1.2, v=0.0600)
    report_progress()
    set_digital_out(0, False)
    new_pose = pose_trans(tuft_coords, p[0.9279, 0.8486, 0.1500, 0, 0, 0])
    movel(p[new_pose[0], new_pose[1], new_pose[2], current_pose[3], current_pose[4], current_pose[5]], a=0.8, v=0.2000)
    report_progress()
    new_pose = pose_trans(tuft_coords, p[0.9299, 0.2034, 0.1500, 0, 0, 0])
    movel(p[new_pose[0], new_pose[1], new_pose[2], current_pose[3], current_pose[4], current_pose[5]], a=1.2, v=0.2000)
    report_progress()
    new_pose = pose_trans(tuft_coords, p[0.9299, 0.2034, -0.0020, 0, 0, 0])
    movel(p[new_pose[0], new_pose[1], new_pose[2], current_pose[3], current_pose[4], current_pose[5]], a=0.8, v=0.2000)
    report_progress()
    set_digital_out(0, True)
    new_pose = pose_trans(tuft_coords, p[0.9299, 0.8466, -0.0020, 0, 0, 0])
    movel(p[new_pose[0], new_pose[1], new_pose[2], current_pose[3], current_pose[4], current_pose[5]], a=1.2, v=0.0600)
    report_progress()
    set_digital_out(0, False)
    new_pose = pose_trans(tuft_coords, p[0.9299, 0.8466, 0.1500, 0, 0, 0])
    movel(p[new_pose[0], new_pose[1], new_pose[2], current_pose[3], current_pose[4], current_pose[5]], a=0.8, v=0.2000)
    report_progress()
    new_pose = pose_trans(tuft_coords, p[0.9318, 0.2034, 0.1500, 0, 0, 0])
    movel(p[new_pose[0], new_pose[1], new_pose[2], current_pose[3], current_pose[4], current_pose[5]], a=1.2, v=0.2000)
    report_progress()
    new_pose = pose_trans(tuft_coords, p[0.9318, 0.2034, -0.0020, 0, 0, 0])
    movel(p[new_pose[0], new_pose[1], new_pose[2], current_pose[3], current_pose[4], current_pose[5]], a=0.8, v=0.2000)
    report_progress()
    set_digital_out(0, True)
    new_pose = pose_trans(tuft_coords, p[0.9318, 0.8466, -0.0020, 0, 0, 0])
    movel(p[new_pose[0], new_pose[1], new_pose[2], current_pose[3], current_pose[4], current_pose[5]], a=1.2, v=0.0600)
    report_progress()
    set_digital_out(0, False)
    new_pose = pose_trans(tuft_coords, p[0.9318, 0.8466, 0.1500, 0, 0, 0])
    movel(p[new_pose[0], new_pose[1], new_pose[2], current_pose[3], current_pose[4], current_pose[5]], a=0.8, v=0.2000)
    report_progress()
    new_pose = pose_trans(tuft_coords, p[0.9337, 0.2054, 0.1500, 0, 0, 0])
    movel(p[new_pose[0], new_pose[1], new_pose[2], current_pose[3], current_pose[4], current_pose[5]], a=1.2, v=0.2000)
    report_progress()
    new_pose = pose_trans(tuft_coords, p[0.9337, 0.2054, -0.0020, 0, 0, 0])
    movel(p[new_pose[0], new_pose[1], new_pose[2], current_pose[3], current_pose[4], current_pose[5]], a=0.8, v=0.2000)
    report_progress()
    set_digital_out(0, True)
    new_pose = pose_trans(tuft_coords, p[0.9337, 0.8446, -0.0020, 0, 0, 0])
    movel(p[new_pose[0], new_pose[1], new_pose[2], current_pose[3], current_pose[4], current_pose[5]], a=1.2, v=0.0600)
    report_progress()
    set_digital_out(0, False)
    new_pose = pose_trans(tuft_coords, p[0.9337, 0.8446, 0.1500, 0, 0, 0])
    movel(p[new_pose[0], new_pose[1], new_pose[2], current_pose[3], current_pose[4], current_pose[5]], a=0.8, v=0.2000)
    report_progress()
    new_pose = pose_trans(tuft_coords, p[0.9357, 0.2054, 0.1500, 0, 0, 0])
    movel(p[new_pose[0], new_pose[1], new_pose[2], current_pose[3], current_pose[4], current_pose[5]], a=1.2, v=0.2000)
    report_progress()
    new_pose = pose_trans(tuft_coords, p[0.9357, 0.2054, -0.0020, 0, 0, 0])
    movel(p[new_pose[0], new_pose[1], new_pose[2], current_pose[3], current_pose[4], current_pose[5]], a=0.8, v=0.2000)
    report_progress()
    set_digital_out(0, True)
    new_pose = pose_trans(tuft_coords, p[0.9357, 0.8446, -0.0020, 0, 0, 0])
    movel(p[new_pose[0], new_pose[1], new_pose[2], current_pose[3], current_pose[4], current_pose[5]], a=1.2, v=0.0600)
    report_progress()
    set_digital_out(0, False)
    new_pose = pose_trans(tuft_coords, p[0.9357, 0.8446, 0.1500, 0, 0, 0])
    movel(p[new_pose[0], new_pose[1], new_pose[2], current_pose[3], current_pose[4], current_pose[5]], a=0.8, v=0.2000)
    report_progress()
    new_pose = pose_trans(tuft_coords, p[0.9376, 0.2073, 0.1500, 0, 0, 0])
    movel(p[new_pose[0], new_pose[1], new_pose[2], current_pose[3], current_pose[4], current_pose[5]], a=1.2, v=0.2000)
    report_progress()
    new_pose = pose_trans(tuft_coords, p[0.9376, 0.2073, -0.0020, 0, 0, 0])
    movel(p[new_pose[0], new_pose[1], new_pose[2], current_pose[3], current_pose[4], current_pose[5]], a=0.8, v=0.2000)
    report_progress()
    set_digital_out(0, True)
    new_pose = pose_trans(tuft_coords, p[0.9376, 0.8427, -0.0020, 0, 0, 0])
    movel(p[new_pose[0], new_pose[1], new_pose[2], current_pose[3], current_pose[4], current_pose[5]], a=1.2, v=0.0600)
    report_progress()
    set_digital_out(0, False)
    new_pose = pose_trans(tuft_coords, p[0.9376, 0.8427, 0.1500, 0, 0, 0])
    movel(p[new_pose[0], new_pose[1], new_pose[2], current_pose[3], current_pose[4], current_pose[5]], a=0.8, v=0.2000)
    report_progress()
    new_pose = pose_trans(tuft_coords, p[0.9396, 0.2093, 0.1500, 0, 0, 0])
    movel(p[new_pose[0], new_pose[1], new_pose[2], current_pose[3], current_pose[4], current_pose[5]], a=1.2, v=0.2000)
    report_progress()
    new_pose = pose_trans(tuft_coords, p[0.9396, 0.2093, -0.0020, 0, 0, 0])
    movel(p[new_pose[0], new_pose[1], new_pose[2], current_pose[3], current_pose[4], current_pose[5]], a=0.8, v=0.2000)
    report_progress()
    set_digital_out(0, True)
    new_pose = pose_trans(tuft_coords, p[0.9396, 0.8407, -0.0020, 0, 0, 0])
    movel(p[new_pose[0], new_pose[1], new_pose[2], current_pose[3], current_pose[4], current_pose[5]], a=1.2, v=0.0600)
    report_progress()
    set_digital_out(0, False)
    new_pose = pose_trans(tuft_coords, p[0.9396, 0.8407, 0.1500, 0, 0, 0])
    movel(p[new_pose[0], new_pose[1], new_pose[2], current_pose[3], current_pose[4], current_pose[5]], a=0.8, v=0.2000)
    report_progress()
    new_pose = pose_trans(tuft_coords, p[0.9415, 0.2093, 0.1500, 0, 0, 0])
    movel(p[new_pose[0], new_pose[1], new_pose[2], current_pose[3], current_pose[4], current_pose[5]], a=1.2, v=0.2000)
    report_progress()
    new_pose = pose_trans(tuft_coords, p[0.9415, 0.2093, -0.0020, 0, 0, 0])
    movel(p[new_pose[0], new_pose[1], new_pose[2], current_pose[3], current_pose[4], current_pose[5]], a=0.8, v=0.2000)
    report_progress()
    set_digital_out(0, True)
    new_pose = pose_trans(tuft_coords, p[0.9415, 0.8407, -0.0020, 0, 0, 0])
    movel(p[new_pose[0], new_pose[1], new_pose[2], current_pose[3], current_pose[4], current_pose[5]], a=1.2, v=0.0600)
    report_progress()
    set_digital_out(0, False)
    new_pose = pose_trans(tuft_coords, p[0.9415, 0.8407, 0.1500, 0, 0, 0])
    movel(p[new_pose[0], new_pose[1], new_pose[2], current_pose[3], current_pose[4], current_pose[5]], a=0.8, v=0.2000)
    report_progress()
    new_pose = pose_trans(tuft_coords, p[0.9435, 0.2113, 0.1500, 0, 0, 0])
    movel(p[new_pose[0], new_pose[1], new_pose[2], current_pose[3], current_pose[4], current_pose[5]], a=1.2, v=0.2000)
    report_progress()
    new_pose = pose_trans(tuft_coords, p[0.9435, 0.2113, -0.0020, 0, 0, 0])
    movel(p[new_pose[0], new_pose[1], new_pose[2], current_pose[3], current_pose[4], current_pose[5]], a=0.8, v=0.2000)
    report_progress()
    set_digital_out(0, True)
    new_pose = pose_trans(tuft_coords, p[0.9435, 0.8387, -0.0020, 0, 0, 0])
    movel(p[new_pose[0], new_pose[1], new_pose[2], current_pose[3], current_pose[4], current_pose[5]], a=1.2, v=0.0600)
    report_progress()
    set_digital_out(0, False)
    new_pose = pose_trans(tuft_coords, p[0.9435, 0.8387, 0.1500, 0, 0, 0])
    movel(p[new_pose[0], new_pose[1], new_pose[2], current_pose[3], current_pose[4], current_pose[5]], a=0.8, v=0.2000)
    report_progress()
    new_pose = pose_trans(tuft_coords, p[0.9454, 0.2113, 0.1500, 0, 0, 0])
    movel(p[new_pose[0], new_pose[1], new_pose[2], current_pose[3], current_pose[4], current_pose[5]], a=1.2, v=0.2000)
    report_progress()
    new_pose = pose_trans(tuft_coords, p[0.9454, 0.2113, -0.0020, 0, 0, 0])
    movel(p[new_pose[0], new_pose[1], new_pose[2], current_pose[3], current_pose[4], current_pose[5]], a=0.8, v=0.2000)
    report_progress()
    set_digital_out(0, True)
    new_pose = pose_trans(tuft_coords, p[0.9454, 0.8387, -0.0020, 0, 0, 0])
    movel(p[new_pose[0], new_pose[1], new_pose[2], current_pose[3], current_pose[4], current_pose[5]], a=1.2, v=0.0600)
    report_progress()
    set_digital_out(0, False)
    new_pose = pose_trans(tuft_coords, p[0.9454, 0.8387, 0.1500, 0, 0, 0])
    movel(p[new_pose[0], new_pose[1], new_pose[2], current_pose[3], current_pose[4], current_pose[5]], a=0.8, v=0.2000)
    report_progress()
    new_pose = pose_trans(tuft_coords, p[0.9474, 0.2133, 0.1500, 0, 0, 0])
    movel(p[new_pose[0], new_pose[1], new_pose[2], current_pose[3], current_pose[4], current_pose[5]], a=1.2, v=0.2000)
    report_progress()
    new_pose = pose_trans(tuft_coords, p[0.9474, 0.2133, -0.0020, 0, 0, 0])
    movel(p[new_pose[0], new_pose[1], new_pose[2], current_pose[3], current_pose[4], current_pose[5]], a=0.8, v=0.2000)
    report_progress()
    set_digital_out(0, True)
    new_pose = pose_trans(tuft_coords, p[0.9474, 0.8367, -0.0020, 0, 0, 0])
    movel(p[new_pose[0], new_pose[1], new_pose[2], current_pose[3], current_pose[4], current_pose[5]], a=1.2, v=0.0600)
    report_progress()
    set_digital_out(0, False)
    new_pose = pose_trans(tuft_coords, p[0.9474, 0.8367, 0.1500, 0, 0, 0])
    movel(p[new_pose[0], new_pose[1], new_pose[2], current_pose[3], current_pose[4], current_pose[5]], a=0.8, v=0.2000)
    report_progress()
    new_pose = pose_trans(tuft_coords, p[0.9493, 0.2153, 0.1500, 0, 0, 0])
    movel(p[new_pose[0], new_pose[1], new_pose[2], current_pose[3], current_pose[4], current_pose[5]], a=1.2, v=0.2000)
    report_progress()
    new_pose = pose_trans(tuft_coords, p[0.9493, 0.2153, -0.0020, 0, 0, 0])
    movel(p[new_pose[0], new_pose[1], new_pose[2], current_pose[3], current_pose[4], current_pose[5]], a=0.8, v=0.2000)
    report_progress()
    set_digital_out(0, True)
    new_pose = pose_trans(tuft_coords, p[0.9493, 0.8347, -0.0020, 0, 0, 0])
    movel(p[new_pose[0], new_pose[1], new_pose[2], current_pose[3], current_pose[4], current_pose[5]], a=1.2, v=0.0600)
    report_progress()
    set_digital_out(0, False)
    new_pose = pose_trans(tuft_coords, p[0.9493, 0.8347, 0.1500, 0, 0, 0])
    movel(p[new_pose[0], new_pose[1], new_pose[2], current_pose[3], current_pose[4], current_pose[5]], a=0.8, v=0.2000)
    report_progress()
    new_pose = pose_trans(tuft_coords, p[0.9513, 0.2153, 0.1500, 0, 0, 0])
    movel(p[new_pose[0], new_pose[1], new_pose[2], current_pose[3], current_pose[4], current_pose[5]], a=1.2, v=0.2000)
    report_progress()
    new_pose = pose_trans(tuft_coords, p[0.9513, 0.2153, -0.0020, 0, 0, 0])
    movel(p[new_pose[0], new_pose[1], new_pose[2], current_pose[3], current_pose[4], current_pose[5]], a=0.8, v=0.2000)
    report_progress()
    set_digital_out(0, True)
    new_pose = pose_trans(tuft_coords, p[0.9513, 0.8347, -0.0020, 0, 0, 0])
    movel(p[new_pose[0], new_pose[1], new_pose[2], current_pose[3], current_pose[4], current_pose[5]], a=1.2, v=0.0600)
    report_progress()
    set_digital_out(0, False)
    new_pose = pose_trans(tuft_coords, p[0.9513, 0.8347, 0.1500, 0, 0, 0])
    movel(p[new_pose[0], new_pose[1], new_pose[2], current_pose[3], current_pose[4], current_pose[5]], a=0.8, v=0.2000)
    report_progress()
    new_pose = pose_trans(tuft_coords, p[0.9532, 0.2172, 0.1500, 0, 0, 0])
    movel(p[new_pose[0], new_pose[1], new_pose[2], current_pose[3], current_pose[4], current_pose[5]], a=1.2, v=0.2000)
    report_progress()
    new_pose = pose_trans(tuft_coords, p[0.9532, 0.2172, -0.0020, 0, 0, 0])
    movel(p[new_pose[0], new_pose[1], new_pose[2], current_pose[3], current_pose[4], current_pose[5]], a=0.8, v=0.2000)
    report_progress()
    set_digital_out(0, True)
    new_pose = pose_trans(tuft_coords, p[0.9532, 0.8328, -0.0020, 0, 0, 0])
    movel(p[new_pose[0], new_pose[1], new_pose[2], current_pose[3], current_pose[4], current_pose[5]], a=1.2, v=0.0600)
    report_progress()
    set_digital_out(0, False)
    new_pose = pose_trans(tuft_coords, p[0.9532, 0.8328, 0.1500, 0, 0, 0])
    movel(p[new_pose[0], new_pose[1], new_pose[2], current_pose[3], current_pose[4], current_pose[5]], a=0.8, v=0.2000)
    report_progress()
    new_pose = pose_trans(tuft_coords, p[0.9551, 0.2192, 0.1500, 0, 0, 0])
    movel(p[new_pose[0], new_pose[1], new_pose[2], current_pose[3], current_pose[4], current_pose[5]], a=1.2, v=0.2000)
    report_progress()
    new_pose = pose_trans(tuft_coords, p[0.9551, 0.2192, -0.0020, 0, 0, 0])
    movel(p[new_pose[0], new_pose[1], new_pose[2], current_pose[3], current_pose[4], current_pose[5]], a=0.8, v=0.2000)
    report_progress()
    set_digital_out(0, True)
    new_pose = pose_trans(tuft_coords, p[0.9551, 0.8308, -0.0020, 0, 0, 0])
    movel(p[new_pose[0], new_pose[1], new_pose[2], current_pose[3], current_pose[4], current_pose[5]], a=1.2, v=0.0600)
    report_progress()
    set_digital_out(0, False)
    new_pose = pose_trans(tuft_coords, p[0.9551, 0.8308, 0.1500, 0, 0, 0])
    movel(p[new_pose[0], new_pose[1], new_pose[2], current_pose[3], current_pose[4], current_pose[5]], a=0.8, v=0.2000)
    report_progress()
    new_pose = pose_trans(tuft_coords, p[0.9571, 0.2192, 0.1500, 0, 0, 0])
    movel(p[new_pose[0], new_pose[1], new_pose[2], current_pose[3], current_pose[4], current_pose[5]], a=1.2, v=0.2000)
    report_progress()
    new_pose = pose_trans(tuft_coords, p[0.9571, 0.2192, -0.0020, 0, 0, 0])
    movel(p[new_pose[0], new_pose[1], new_pose[2], current_pose[3], current_pose[4], current_pose[5]], a=0.8, v=0.2000)
    report_progress()
    set_digital_out(0, True)
    new_pose = pose_trans(tuft_coords, p[0.9571, 0.8308, -0.0020, 0, 0, 0])
    movel(p[new_pose[0], new_pose[1], new_pose[2], current_pose[3], current_pose[4], current_pose[5]], a=1.2, v=0.0600)
    report_progress()
    set_digital_out(0, False)
    new_pose = pose_trans(tuft_coords, p[0.9571, 0.8308, 0.1500, 0, 0, 0])
    movel(p[new_pose[0], new_pose[1], new_pose[2], current_pose[3], current_pose[4], current_pose[5]], a=0.8, v=0.2000)
    report_progress()
    new_pose = pose_trans(tuft_coords, p[0.9590, 0.2212, 0.1500, 0, 0, 0])
    movel(p[new_pose[0], new_pose[1], new_pose[2], current_pose[3], current_pose[4], current_pose[5]], a=1.2, v=0.2000)
    report_progress()
    new_pose = pose_trans(tuft_coords, p[0.9590, 0.2212, -0.0020, 0, 0, 0])
    movel(p[new_pose[0], new_pose[1], new_pose[2], current_pose[3], current_pose[4], current_pose[5]], a=0.8, v=0.2000)
    report_progress()
    set_digital_out(0, True)
    new_pose = pose_trans(tuft_coords, p[0.9590, 0.8288, -0.0020, 0, 0, 0])
    movel(p[new_pose[0], new_pose[1], new_pose[2], current_pose[3], current_pose[4], current_pose[5]], a=1.2, v=0.0600)
    report_progress()
    set_digital_out(0, False)
    new_pose = pose_trans(tuft_coords, p[0.9590, 0.8288, 0.1500, 0, 0, 0])
    movel(p[new_pose[0], new_pose[1], new_pose[2], current_pose[3], current_pose[4], current_pose[5]], a=0.8, v=0.2000)
    report_progress()
    new_pose = pose_trans(tuft_coords, p[0.9610, 0.2232, 0.1500, 0, 0, 0])
    movel(p[new_pose[0], new_pose[1], new_pose[2], current_pose[3], current_pose[4], current_pose[5]], a=1.2, v=0.2000)
    report_progress()
    new_pose = pose_trans(tuft_coords, p[0.9610, 0.2232, -0.0020, 0, 0, 0])
    movel(p[new_pose[0], new_pose[1], new_pose[2], current_pose[3], current_pose[4], current_pose[5]], a=0.8, v=0.2000)
    report_progress()
    set_digital_out(0, True)
    new_pose = pose_trans(tuft_coords, p[0.9610, 0.8268, -0.0020, 0, 0, 0])
    movel(p[new_pose[0], new_pose[1], new_pose[2], current_pose[3], current_pose[4], current_pose[5]], a=1.2, v=0.0600)
    report_progress()
    set_digital_out(0, False)
    new_pose = pose_trans(tuft_coords, p[0.9610, 0.8268, 0.1500, 0, 0, 0])
    movel(p[new_pose[0], new_pose[1], new_pose[2], current_pose[3], current_pose[4], current_pose[5]], a=0.8, v=0.2000)
    report_progress()
    new_pose = pose_trans(tuft_coords, p[0.9629, 0.2232, 0.1500, 0, 0, 0])
    movel(p[new_pose[0], new_pose[1], new_pose[2], current_pose[3], current_pose[4], current_pose[5]], a=1.2, v=0.2000)
    report_progress()
    new_pose = pose_trans(tuft_coords, p[0.9629, 0.2232, -0.0020, 0, 0, 0])
    movel(p[new_pose[0], new_pose[1], new_pose[2], current_pose[3], current_pose[4], current_pose[5]], a=0.8, v=0.2000)
    report_progress()
    set_digital_out(0, True)
    new_pose = pose_trans(tuft_coords, p[0.9629, 0.8268, -0.0020, 0, 0, 0])
    movel(p[new_pose[0], new_pose[1], new_pose[2], current_pose[3], current_pose[4], current_pose[5]], a=1.2, v=0.0600)
    report_progress()
    set_digital_out(0, False)
    new_pose = pose_trans(tuft_coords, p[0.9629, 0.8268, 0.1500, 0, 0, 0])
    movel(p[new_pose[0], new_pose[1], new_pose[2], current_pose[3], current_pose[4], current_pose[5]], a=0.8, v=0.2000)
    report_progress()
    new_pose = pose_trans(tuft_coords, p[0.9649, 0.2252, 0.1500, 0, 0, 0])
    movel(p[new_pose[0], new_pose[1], new_pose[2], current_pose[3], current_pose[4], current_pose[5]], a=1.2, v=0.2000)
    report_progress()
    new_pose = pose_trans(tuft_coords, p[0.9649, 0.2252, -0.0020, 0, 0, 0])
    movel(p[new_pose[0], new_pose[1], new_pose[2], current_pose[3], current_pose[4], current_pose[5]], a=0.8, v=0.2000)
    report_progress()
    set_digital_out(0, True)
    new_pose = pose_trans(tuft_coords, p[0.9649, 0.8248, -0.0020, 0, 0, 0])
    movel(p[new_pose[0], new_pose[1], new_pose[2], current_pose[3], current_pose[4], current_pose[5]], a=1.2, v=0.0600)
    report_progress()
    set_digital_out(0, False)
    new_pose = pose_trans(tuft_coords, p[0.9649, 0.8248, 0.1500, 0, 0, 0])
    movel(p[new_pose[0], new_pose[1], new_pose[2], current_pose[3], current_pose[4], current_pose[5]], a=0.8, v=0.2000)
    report_progress()
    new_pose = pose_trans(tuft_coords, p[0.9668, 0.2271, 0.1500, 0, 0, 0])
    movel(p[new_pose[0], new_pose[1], new_pose[2], current_pose[3], current_pose[4], current_pose[5]], a=1.2, v=0.2000)
    report_progress()
    new_pose = pose_trans(tuft_coords, p[0.9668, 0.2271, -0.0020, 0, 0, 0])
    movel(p[new_pose[0], new_pose[1], new_pose[2], current_pose[3], current_pose[4], current_pose[5]], a=0.8, v=0.2000)
    report_progress()
    set_digital_out(0, True)
    new_pose = pose_trans(tuft_coords, p[0.9668, 0.8229, -0.0020, 0, 0, 0])
    movel(p[new_pose[0], new_pose[1], new_pose[2], current_pose[3], current_pose[4], current_pose[5]], a=1.2, v=0.0600)
    report_progress()
    set_digital_out(0, False)
    new_pose = pose_trans(tuft_coords, p[0.9668, 0.8229, 0.1500, 0, 0, 0])
    movel(p[new_pose[0], new_pose[1], new_pose[2], current_pose[3], current_pose[4], current_pose[5]], a=0.8, v=0.2000)
    report_progress()
    new_pose = pose_trans(tuft_coords, p[0.9688, 0.2291, 0.1500, 0, 0, 0])
    movel(p[new_pose[0], new_pose[1], new_pose[2], current_pose[3], current_pose[4], current_pose[5]], a=1.2, v=0.2000)
    report_progress()
    new_pose = pose_trans(tuft_coords, p[0.9688, 0.2291, -0.0020, 0, 0, 0])
    movel(p[new_pose[0], new_pose[1], new_pose[2], current_pose[3], current_pose[4], current_pose[5]], a=0.8, v=0.2000)
    report_progress()
    set_digital_out(0, True)
    new_pose = pose_trans(tuft_coords, p[0.9688, 0.8209, -0.0020, 0, 0, 0])
    movel(p[new_pose[0], new_pose[1], new_pose[2], current_pose[3], current_pose[4], current_pose[5]], a=1.2, v=0.0600)
    report_progress()
    set_digital_out(0, False)
    new_pose = pose_trans(tuft_coords, p[0.9688, 0.8209, 0.1500, 0, 0, 0])
    movel(p[new_pose[0], new_pose[1], new_pose[2], current_pose[3], current_pose[4], current_pose[5]], a=0.8, v=0.2000)
    report_progress()
    new_pose = pose_trans(tuft_coords, p[0.9707, 0.2291, 0.1500, 0, 0, 0])
    movel(p[new_pose[0], new_pose[1], new_pose[2], current_pose[3], current_pose[4], current_pose[5]], a=1.2, v=0.2000)
    report_progress()
    new_pose = pose_trans(tuft_coords, p[0.9707, 0.2291, -0.0020, 0, 0, 0])
    movel(p[new_pose[0], new_pose[1], new_pose[2], current_pose[3], current_pose[4], current_pose[5]], a=0.8, v=0.2000)
    report_progress()
    set_digital_out(0, True)
    new_pose = pose_trans(tuft_coords, p[0.9707, 0.8209, -0.0020, 0, 0, 0])
    movel(p[new_pose[0], new_pose[1], new_pose[2], current_pose[3], current_pose[4], current_pose[5]], a=1.2, v=0.0600)
    report_progress()
    set_digital_out(0, False)
    new_pose = pose_trans(tuft_coords, p[0.9707, 0.8209, 0.1500, 0, 0, 0])
    movel(p[new_pose[0], new_pose[1], new_pose[2], current_pose[3], current_pose[4], current_pose[5]], a=0.8, v=0.2000)
    report_progress()
    new_pose = pose_trans(tuft_coords, p[0.9726, 0.2311, 0.1500, 0, 0, 0])
    movel(p[new_pose[0], new_pose[1], new_pose[2], current_pose[3], current_pose[4], current_pose[5]], a=1.2, v=0.2000)
    report_progress()
    new_pose = pose_trans(tuft_coords, p[0.9726, 0.2311, -0.0020, 0, 0, 0])
    movel(p[new_pose[0], new_pose[1], new_pose[2], current_pose[3], current_pose[4], current_pose[5]], a=0.8, v=0.2000)
    report_progress()
    set_digital_out(0, True)
    new_pose = pose_trans(tuft_coords, p[0.9726, 0.8189, -0.0020, 0, 0, 0])
    movel(p[new_pose[0], new_pose[1], new_pose[2], current_pose[3], current_pose[4], current_pose[5]], a=1.2, v=0.0600)
    report_progress()
    set_digital_out(0, False)
    new_pose = pose_trans(tuft_coords, p[0.9726, 0.8189, 0.1500, 0, 0, 0])
    movel(p[new_pose[0], new_pose[1], new_pose[2], current_pose[3], current_pose[4], current_pose[5]], a=0.8, v=0.2000)
    report_progress()
    new_pose = pose_trans(tuft_coords, p[0.9746, 0.2331, 0.1500, 0, 0, 0])
    movel(p[new_pose[0], new_pose[1], new_pose[2], current_pose[3], current_pose[4], current_pose[5]], a=1.2, v=0.2000)
    report_progress()
    new_pose = pose_trans(tuft_coords, p[0.9746, 0.2331, -0.0020, 0, 0, 0])
    movel(p[new_pose[0], new_pose[1], new_pose[2], current_pose[3], current_pose[4], current_pose[5]], a=0.8, v=0.2000)
    report_progress()
    set_digital_out(0, True)
    new_pose = pose_trans(tuft_coords, p[0.9746, 0.8169, -0.0020, 0, 0, 0])
    movel(p[new_pose[0], new_pose[1], new_pose[2], current_pose[3], current_pose[4], current_pose[5]], a=1.2, v=0.0600)
    report_progress()
    set_digital_out(0, False)
    new_pose = pose_trans(tuft_coords, p[0.9746, 0.8169, 0.1500, 0, 0, 0])
    movel(p[new_pose[0], new_pose[1], new_pose[2], current_pose[3], current_pose[4], current_pose[5]], a=0.8, v=0.2000)
    report_progress()
    new_pose = pose_trans(tuft_coords, p[0.9765, 0.2351, 0.1500, 0, 0, 0])
    movel(p[new_pose[0], new_pose[1], new_pose[2], current_pose[3], current_pose[4], current_pose[5]], a=1.2, v=0.2000)
    report_progress()
    new_pose = pose_trans(tuft_coords, p[0.9765, 0.2351, -0.0020, 0, 0, 0])
    movel(p[new_pose[0], new_pose[1], new_pose[2], current_pose[3], current_pose[4], current_pose[5]], a=0.8, v=0.2000)
    report_progress()
    set_digital_out(0, True)
    new_pose = pose_trans(tuft_coords, p[0.9765, 0.8149, -0.0020, 0, 0, 0])
    movel(p[new_pose[0], new_pose[1], new_pose[2], current_pose[3], current_pose[4], current_pose[5]], a=1.2, v=0.0600)
    report_progress()
    set_digital_out(0, False)
    new_pose = pose_trans(tuft_coords, p[0.9765, 0.8149, 0.1500, 0, 0, 0])
    movel(p[new_pose[0], new_pose[1], new_pose[2], current_pose[3], current_pose[4], current_pose[5]], a=0.8, v=0.2000)
    report_progress()
    new_pose = pose_trans(tuft_coords, p[0.9785, 0.2351, 0.1500, 0, 0, 0])
    movel(p[new_pose[0], new_pose[1], new_pose[2], current_pose[3], current_pose[4], current_pose[5]], a=1.2, v=0.2000)
    report_progress()
    new_pose = pose_trans(tuft_coords, p[0.9785, 0.2351, -0.0020, 0, 0, 0])
    movel(p[new_pose[0], new_pose[1], new_pose[2], current_pose[3], current_pose[4], current_pose[5]], a=0.8, v=0.2000)
    report_progress()
    set_digital_out(0, True)
    new_pose = pose_trans(tuft_coords, p[0.9785, 0.8149, -0.0020, 0, 0, 0])
    movel(p[new_pose[0], new_pose[1], new_pose[2], current_pose[3], current_pose[4], current_pose[5]], a=1.2, v=0.0600)
    report_progress()
    set_digital_out(0, False)
    new_pose = pose_trans(tuft_coords, p[0.9785, 0.8149, 0.1500, 0, 0, 0])
    movel(p[new_pose[0], new_pose[1], new_pose[2], current_pose[3], current_pose[4], current_pose[5]], a=0.8, v=0.2000)
    report_progress()
    new_pose = pose_trans(tuft_coords, p[0.9804, 0.2370, 0.1500, 0, 0, 0])
    movel(p[new_pose[0], new_pose[1], new_pose[2], current_pose[3], current_pose[4], current_pose[5]], a=1.2, v=0.2000)
    report_progress()
    new_pose = pose_trans(tuft_coords, p[0.9804, 0.2370, -0.0020, 0, 0, 0])
    movel(p[new_pose[0], new_pose[1], new_pose[2], current_pose[3], current_pose[4], current_pose[5]], a=0.8, v=0.2000)
    report_progress()
    set_digital_out(0, True)
    new_pose = pose_trans(tuft_coords, p[0.9804, 0.8130, -0.0020, 0, 0, 0])
    movel(p[new_pose[0], new_pose[1], new_pose[2], current_pose[3], current_pose[4], current_pose[5]], a=1.2, v=0.0600)
    report_progress()
    set_digital_out(0, False)
    new_pose = pose_trans(tuft_coords, p[0.9804, 0.8130, 0.1500, 0, 0, 0])
    movel(p[new_pose[0], new_pose[1], new_pose[2], current_pose[3], current_pose[4], current_pose[5]], a=0.8, v=0.2000)
    report_progress()
    new_pose = pose_trans(tuft_coords, p[0.9824, 0.2390, 0.1500, 0, 0, 0])
    movel(p[new_pose[0], new_pose[1], new_pose[2], current_pose[3], current_pose[4], current_pose[5]], a=1.2, v=0.2000)
    report_progress()
    new_pose = pose_trans(tuft_coords, p[0.9824, 0.2390, -0.0020, 0, 0, 0])
    movel(p[new_pose[0], new_pose[1], new_pose[2], current_pose[3], current_pose[4], current_pose[5]], a=0.8, v=0.2000)
    report_progress()
    set_digital_out(0, True)
    new_pose = pose_trans(tuft_coords, p[0.9824, 0.8110, -0.0020, 0, 0, 0])
    movel(p[new_pose[0], new_pose[1], new_pose[2], current_pose[3], current_pose[4], current_pose[5]], a=1.2, v=0.0600)
    report_progress()
    set_digital_out(0, False)
    new_pose = pose_trans(tuft_coords, p[0.9824, 0.8110, 0.1500, 0, 0, 0])
    movel(p[new_pose[0], new_pose[1], new_pose[2], current_pose[3], current_pose[4], current_pose[5]], a=0.8, v=0.2000)
    report_progress()
    new_pose = pose_trans(tuft_coords, p[0.9843, 0.2410, 0.1500, 0, 0, 0])
    movel(p[new_pose[0], new_pose[1], new_pose[2], current_pose[3], current_pose[4], current_pose[5]], a=1.2, v=0.2000)
    report_progress()
    new_pose = pose_trans(tuft_coords, p[0.9843, 0.2410, -0.0020, 0, 0, 0])
    movel(p[new_pose[0], new_pose[1], new_pose[2], current_pose[3], current_pose[4], current_pose[5]], a=0.8, v=0.2000)
    report_progress()
    set_digital_out(0, True)
    new_pose = pose_trans(tuft_coords, p[0.9843, 0.8090, -0.0020, 0, 0, 0])
    movel(p[new_pose[0], new_pose[1], new_pose[2], current_pose[3], current_pose[4], current_pose[5]], a=1.2, v=0.0600)
    report_progress()
    set_digital_out(0, False)
    new_pose = pose_trans(tuft_coords, p[0.9843, 0.8090, 0.1500, 0, 0, 0])
    movel(p[new_pose[0], new_pose[1], new_pose[2], current_pose[3], current_pose[4], current_pose[5]], a=0.8, v=0.2000)
    report_progress()
    new_pose = pose_trans(tuft_coords, p[0.9862, 0.2430, 0.1500, 0, 0, 0])
    movel(p[new_pose[0], new_pose[1], new_pose[2], current_pose[3], current_pose[4], current_pose[5]], a=1.2, v=0.2000)
    report_progress()
    new_pose = pose_trans(tuft_coords, p[0.9862, 0.2430, -0.0020, 0, 0, 0])
    movel(p[new_pose[0], new_pose[1], new_pose[2], current_pose[3], current_pose[4], current_pose[5]], a=0.8, v=0.2000)
    report_progress()
    set_digital_out(0, True)
    new_pose = pose_trans(tuft_coords, p[0.9862, 0.8070, -0.0020, 0, 0, 0])
    movel(p[new_pose[0], new_pose[1], new_pose[2], current_pose[3], current_pose[4], current_pose[5]], a=1.2, v=0.0600)
    report_progress()
    set_digital_out(0, False)
    new_pose = pose_trans(tuft_coords, p[0.9862, 0.8070, 0.1500, 0, 0, 0])
    movel(p[new_pose[0], new_pose[1], new_pose[2], current_pose[3], current_pose[4], current_pose[5]], a=0.8, v=0.2000)
    report_progress()
    new_pose = pose_trans(tuft_coords, p[0.9882, 0.2449, 0.1500, 0, 0, 0])
    movel(p[new_pose[0], new_pose[1], new_pose[2], current_pose[3], current_pose[4], current_pose[5]], a=1.2, v=0.2000)
    report_progress()
    new_pose = pose_trans(tuft_coords, p[0.9882, 0.2449, -0.0020, 0, 0, 0])
    movel(p[new_pose[0], new_pose[1], new_pose[2], current_pose[3], current_pose[4], current_pose[5]], a=0.8, v=0.2000)
    report_progress()
    set_digital_out(0, True)
    new_pose = pose_trans(tuft_coords, p[0.9882, 0.8051, -0.0020, 0, 0, 0])
    movel(p[new_pose[0], new_pose[1], new_pose[2], current_pose[3], current_pose[4], current_pose[5]], a=1.2, v=0.0600)
    report_progress()
    set_digital_out(0, False)
    new_pose = pose_trans(tuft_coords, p[0.9882, 0.8051, 0.1500, 0, 0, 0])
    movel(p[new_pose[0], new_pose[1], new_pose[2], current_pose[3], current_pose[4], current_pose[5]], a=0.8, v=0.2000)
    report_progress()
    new_pose = pose_trans(tuft_coords, p[0.9901, 0.2469, 0.1500, 0, 0, 0])
    movel(p[new_pose[0], new_pose[1], new_pose[2], current_pose[3], current_pose[4], current_pose[5]], a=1.2, v=0.2000)
    report_progress()
    new_pose = pose_trans(tuft_coords, p[0.9901, 0.2469, -0.0020, 0, 0, 0])
    movel(p[new_pose[0], new_pose[1], new_pose[2], current_pose[3], current_pose[4], current_pose[5]], a=0.8, v=0.2000)
    report_progress()
    set_digital_out(0, True)
    new_pose = pose_trans(tuft_coords, p[0.9901, 0.8031, -0.0020, 0, 0, 0])
    movel(p[new_pose[0], new_pose[1], new_pose[2], current_pose[3], current_pose[4], current_pose[5]], a=1.2, v=0.0600)
    report_progress()
    set_digital_out(0, False)
    new_pose = pose_trans(tuft_coords, p[0.9901, 0.8031, 0.1500, 0, 0, 0])
    movel(p[new_pose[0], new_pose[1], new_pose[2], current_pose[3], current_pose[4], current_pose[5]], a=0.8, v=0.2000)
    report_progress()
    new_pose = pose_trans(tuft_coords, p[0.9921, 0.2469, 0.1500, 0, 0, 0])
    movel(p[new_pose[0], new_pose[1], new_pose[2], current_pose[3], current_pose[4], current_pose[5]], a=1.2, v=0.2000)
    report_progress()
    new_pose = pose_trans(tuft_coords, p[0.9921, 0.2469, -0.0020, 0, 0, 0])
    movel(p[new_pose[0], new_pose[1], new_pose[2], current_pose[3], current_pose[4], current_pose[5]], a=0.8, v=0.2000)
    report_progress()
    set_digital_out(0, True)
    new_pose = pose_trans(tuft_coords, p[0.9921, 0.8031, -0.0020, 0, 0, 0])
    movel(p[new_pose[0], new_pose[1], new_pose[2], current_pose[3], current_pose[4], current_pose[5]], a=1.2, v=0.0600)
    report_progress()
    set_digital_out(0, False)
    new_pose = pose_trans(tuft_coords, p[0.9921, 0.8031, 0.1500, 0, 0, 0])
    movel(p[new_pose[0], new_pose[1], new_pose[2], current_pose[3], current_pose[4], current_pose[5]], a=0.8, v=0.2000)
    report_progress()
    new_pose = pose_trans(tuft_coords, p[0.9940, 0.2489, 0.1500, 0, 0, 0])
    movel(p[new_pose[0], new_pose[1], new_pose[2], current_pose[3], current_pose[4], current_pose[5]], a=1.2, v=0.2000)
    report_progress()
    new_pose = pose_trans(tuft_coords, p[0.9940, 0.2489, -0.0020, 0, 0, 0])
    movel(p[new_pose[0], new_pose[1], new_pose[2], current_pose[3], current_pose[4], current_pose[5]], a=0.8, v=0.2000)
    report_progress()
    set_digital_out(0, True)
    new_pose = pose_trans(tuft_coords, p[0.9940, 0.8011, -0.0020, 0, 0, 0])
    movel(p[new_pose[0], new_pose[1], new_pose[2], current_pose[3], current_pose[4], current_pose[5]], a=1.2, v=0.0600)
    report_progress()
    set_digital_out(0, False)
    new_pose = pose_trans(tuft_coords, p[0.9940, 0.8011, 0.1500, 0, 0, 0])
    movel(p[new_pose[0], new_pose[1], new_pose[2], current_pose[3], current_pose[4], current_pose[5]], a=0.8, v=0.2000)
    report_progress()
    new_pose = pose_trans(tuft_coords, p[0.9960, 0.2509, 0.1500, 0, 0, 0])
    movel(p[new_pose[0], new_pose[1], new_pose[2], current_pose[3], current_pose[4], current_pose[5]], a=1.2, v=0.2000)
    report_progress()
    new_pose = pose_trans(tuft_coords, p[0.9960, 0.2509, -0.0020, 0, 0, 0])
    movel(p[new_pose[0], new_pose[1], new_pose[2], current_pose[3], current_pose[4], current_pose[5]], a=0.8, v=0.2000)
    report_progress()
    set_digital_out(0, True)
    new_pose = pose_trans(tuft_coords, p[0.9960, 0.7991, -0.0020, 0, 0, 0])
    movel(p[new_pose[0], new_pose[1], new_pose[2], current_pose[3], current_pose[4], current_pose[5]], a=1.2, v=0.0600)
    report_progress()
    set_digital_out(0, False)
    new_pose = pose_trans(tuft_coords, p[0.9960, 0.7991, 0.1500, 0, 0, 0])
    movel(p[new_pose[0], new_pose[1], new_pose[2], current_pose[3], current_pose[4], current_pose[5]], a=0.8, v=0.2000)
    report_progress()
    new_pose = pose_trans(tuft_coords, p[0.9979, 0.2529, 0.1500, 0, 0, 0])
    movel(p[new_pose[0], new_pose[1], new_pose[2], current_pose[3], current_pose[4], current_pose[5]], a=1.2, v=0.2000)
    report_progress()
    new_pose = pose_trans(tuft_coords, p[0.9979, 0.2529, -0.0020, 0, 0, 0])
    movel(p[new_pose[0], new_pose[1], new_pose[2], current_pose[3], current_pose[4], current_pose[5]], a=0.8, v=0.2000)
    report_progress()
    set_digital_out(0, True)
    new_pose = pose_trans(tuft_coords, p[0.9979, 0.7971, -0.0020, 0, 0, 0])
    movel(p[new_pose[0], new_pose[1], new_pose[2], current_pose[3], current_pose[4], current_pose[5]], a=1.2, v=0.0600)
    report_progress()
    set_digital_out(0, False)
    new_pose = pose_trans(tuft_coords, p[0.9979, 0.7971, 0.1500, 0, 0, 0])
    movel(p[new_pose[0], new_pose[1], new_pose[2], current_pose[3], current_pose[4], current_pose[5]], a=0.8, v=0.2000)
    report_progress()
    new_pose = pose_trans(tuft_coords, p[0.9999, 0.2548, 0.1500, 0, 0, 0])
    movel(p[new_pose[0], new_pose[1], new_pose[2], current_pose[3], current_pose[4], current_pose[5]], a=1.2, v=0.2000)
    report_progress()
    new_pose = pose_trans(tuft_coords, p[0.9999, 0.2548, -0.0020, 0, 0, 0])
    movel(p[new_pose[0], new_pose[1], new_pose[2], current_pose[3], current_pose[4], current_pose[5]], a=0.8, v=0.2000)
    report_progress()
    set_digital_out(0, True)
    new_pose = pose_trans(tuft_coords, p[0.9999, 0.7952, -0.0020, 0, 0, 0])
    movel(p[new_pose[0], new_pose[1], new_pose[2], current_pose[3], current_pose[4], current_pose[5]], a=1.2, v=0.0600)
    report_progress()
    set_digital_out(0, False)
    new_pose = pose_trans(tuft_coords, p[0.9999, 0.7952, 0.1500, 0, 0, 0])
    movel(p[new_pose[0], new_pose[1], new_pose[2], current_pose[3], current_pose[4], current_pose[5]], a=0.8, v=0.2000)
    report_progress()
    new_pose = pose_trans(tuft_coords, p[1.0018, 0.2568, 0.1500, 0, 0, 0])
    movel(p[new_pose[0], new_pose[1], new_pose[2], current_pose[3], current_pose[4], current_pose[5]], a=1.2, v=0.2000)
    report_progress()
    new_pose = pose_trans(tuft_coords, p[1.0018, 0.2568, -0.0020, 0, 0, 0])
    movel(p[new_pose[0], new_pose[1], new_pose[2], current_pose[3], current_pose[4], current_pose[5]], a=0.8, v=0.2000)
    report_progress()
    set_digital_out(0, True)
    new_pose = pose_trans(tuft_coords, p[1.0018, 0.7932, -0.0020, 0, 0, 0])
    movel(p[new_pose[0], new_pose[1], new_pose[2], current_pose[3], current_pose[4], current_pose[5]], a=1.2, v=0.0600)
    report_progress()
    set_digital_out(0, False)
    new_pose = pose_trans(tuft_coords, p[1.0018, 0.7932, 0.1500, 0, 0, 0])
    movel(p[new_pose[0], new_pose[1], new_pose[2], current_pose[3], current_pose[4], current_pose[5]], a=0.8, v=0.2000)
    report_progress()
    new_pose = pose_trans(tuft_coords, p[1.0037, 0.2588, 0.1500, 0, 0, 0])
    movel(p[new_pose[0], new_pose[1], new_pose[2], current_pose[3], current_pose[4], current_pose[5]], a=1.2, v=0.2000)
    report_progress()
    new_pose = pose_trans(tuft_coords, p[1.0037, 0.2588, -0.0020, 0, 0, 0])
    movel(p[new_pose[0], new_pose[1], new_pose[2], current_pose[3], current_pose[4], current_pose[5]], a=0.8, v=0.2000)
    report_progress()
    set_digital_out(0, True)
    new_pose = pose_trans(tuft_coords, p[1.0037, 0.7912, -0.0020, 0, 0, 0])
    movel(p[new_pose[0], new_pose[1], new_pose[2], current_pose[3], current_pose[4], current_pose[5]], a=1.2, v=0.0600)
    report_progress()
    set_digital_out(0, False)
    new_pose = pose_trans(tuft_coords, p[1.0037, 0.7912, 0.1500, 0, 0, 0])
    movel(p[new_pose[0], new_pose[1], new_pose[2], current_pose[3], current_pose[4], current_pose[5]], a=0.8, v=0.2000)
    report_progress()
    new_pose = pose_trans(tuft_coords, p[1.0057, 0.2608, 0.1500, 0, 0, 0])
    movel(p[new_pose[0], new_pose[1], new_pose[2], current_pose[3], current_pose[4], current_pose[5]], a=1.2, v=0.2000)
    report_progress()
    new_pose = pose_trans(tuft_coords, p[1.0057, 0.2608, -0.0020, 0, 0, 0])
    movel(p[new_pose[0], new_pose[1], new_pose[2], current_pose[3], current_pose[4], current_pose[5]], a=0.8, v=0.2000)
    report_progress()
    set_digital_out(0, True)
    new_pose = pose_trans(tuft_coords, p[1.0057, 0.7892, -0.0020, 0, 0, 0])
    movel(p[new_pose[0], new_pose[1], new_pose[2], current_pose[3], current_pose[4], current_pose[5]], a=1.2, v=0.0600)
    report_progress()
    set_digital_out(0, False)
    new_pose = pose_trans(tuft_coords, p[1.0057, 0.7892, 0.1500, 0, 0, 0])
    movel(p[new_pose[0], new_pose[1], new_pose[2], current_pose[3], current_pose[4], current_pose[5]], a=0.8, v=0.2000)
    report_progress()
    new_pose = pose_trans(tuft_coords, p[1.0076, 0.2628, 0.1500, 0, 0, 0])
    movel(p[new_pose[0], new_pose[1], new_pose[2], current_pose[3], current_pose[4], current_pose[5]], a=1.2, v=0.2000)
    report_progress()
    new_pose = pose_trans(tuft_coords, p[1.0076, 0.2628, -0.0020, 0, 0, 0])
    movel(p[new_pose[0], new_pose[1], new_pose[2], current_pose[3], current_pose[4], current_pose[5]], a=0.8, v=0.2000)
    report_progress()
    set_digital_out(0, True)
    new_pose = pose_trans(tuft_coords, p[1.0076, 0.7872, -0.0020, 0, 0, 0])
    movel(p[new_pose[0], new_pose[1], new_pose[2], current_pose[3], current_pose[4], current_pose[5]], a=1.2, v=0.0600)
    report_progress()
    set_digital_out(0, False)
    new_pose = pose_trans(tuft_coords, p[1.0076, 0.7872, 0.1500, 0, 0, 0])
    movel(p[new_pose[0], new_pose[1], new_pose[2], current_pose[3], current_pose[4], current_pose[5]], a=0.8, v=0.2000)
    report_progress()
    new_pose = pose_trans(tuft_coords, p[1.0096, 0.2647, 0.1500, 0, 0, 0])
    movel(p[new_pose[0], new_pose[1], new_pose[2], current_pose[3], current_pose[4], current_pose[5]], a=1.2, v=0.2000)
    report_progress()
    new_pose = pose_trans(tuft_coords, p[1.0096, 0.2647, -0.0020, 0, 0, 0])
    movel(p[new_pose[0], new_pose[1], new_pose[2], current_pose[3], current_pose[4], current_pose[5]], a=0.8, v=0.2000)
    report_progress()
    set_digital_out(0, True)
    new_pose = pose_trans(tuft_coords, p[1.0096, 0.7853, -0.0020, 0, 0, 0])
    movel(p[new_pose[0], new_pose[1], new_pose[2], current_pose[3], current_pose[4], current_pose[5]], a=1.2, v=0.0600)
